	400: 	// Send mover to the next station
			fMoverPosition     := fNextStationWaitingPosition;
			fMoverVelocity     :=    300.0;
			fMoverAcceleration :=  1_000.0;
			fMoverJerk         := 10_000.0;	
	
			stMoveParameters.direction := Tc3_Mc3PlanarMotion.MC_DIRECTION.mcDirectionPositive;
			stMoveParameters.gap       := 240.0;
			
			strInfo := CONCAT('Station: ', UINT_TO_STRING(nStationIndex));
			strInfo := CONCAT(strInfo, ' Mover: ');
			strInfo := CONCAT(strInfo, UDINT_TO_STRING(nMoverIndex));
			strInfo := CONCAT(strInfo, ' move to next Station:' );
			strInfo := CONCAT(strInfo, UDINT_TO_STRING(nNextStationIndex));
			
		
			IF NOT ipMoverApplication[nMoverIndex].std.P_MoveOnTrack.Busy THEN
	
				FOR idx:=10 TO 1 BY -1 DO 
					strInfoHistory[idx] := strInfoHistory[idx-1];
				END_FOR
				strInfoHistory[0] := strInfo;		
			
				ipMoverApplication[nMoverIndex].std.MoveOnTrack( strInfo,
																 ipTrack[nNextStationTrackIndex].std,
																 fMoverPosition,
																 fMoverVelocity,
																 fMoverAcceleration,
																 fMoverJerk,
																 stMoveParameters.gap,
																 stMoveParameters.direction);
				nStateMoverRecovery := nStateMoverRecovery +1;
				
				
				ipMoverApplication[nMoverIndex].ProductData.bInitRun            := TRUE;
				ipMoverApplication[nMoverIndex].ProductData.nDestinationProcess := 0;
			END_IF	
			
	401: 
		IF ipMoverApplication[nMoverIndex].std.P_MoveOnTrack.Active THEN
			nStateMoverRecovery := 410;
		 END_IF
				 
	410: // Mover to the list of the next station
		ipStation[nNextStationIndex].P_List.AddMover(fbInitList.RemoveFirstInList());
		nStateMoverRecovery := 300;	
	
	500:	// Mover recovery done
			  MoverRecovery := TRUE;
		nStateMoverRecovery := 0;		

END_CASE
END_METHOD

PROPERTY P_bMoverError : BOOL
GET
P_bMoverError := bMoverError;
END_GET
SET
bMoverError := P_bMoverError;
END_SET
END_PROPERTY

PROPERTY PUBLIC P_nAbortingSequence : UDINT
GET
P_nAbortingSequence := nAbortingSequence;
END_GET
END_PROPERTY

PROPERTY PUBLIC P_nExecutingSequence : UDINT
GET
P_nExecutingSequence := nExecutingSequence;
END_GET
END_PROPERTY

PROPERTY PUBLIC P_nResettingSequence : UDINT
GET
P_nResettingSequence := nResettingSequence;
END_GET
END_PROPERTY

PROPERTY PUBLIC P_nStartingSequence : UDINT
GET
P_nStartingSequence := nStartingSequence;
END_GET
END_PROPERTY

PROPERTY PUBLIC P_nStartupSequence : UDINT
GET
P_nStartupSequence := nStartupSequence;
END_GET
END_PROPERTY

METHOD Resetting : BOOL
VAR_INPUT
END_VAR
CASE nResettingSequence OF 
	
	0: //Idle 
		nResettingSequence := 20;
		
		
	20: // Reset Movers
		IF ipMotionSystem.ResetMovers() THEN
			nResettingSequence := 21;
		ELSE
			;// Error			
		END_IF
		
	21: IF ipMotionSystem.P_ResetMovers.Done THEN
			nResettingSequence := 30;
		ELSIF ipMotionSystem.P_ResetMovers.Error THEN
			;//Error 	
		END_IF

		
	30:	nResettingSequence := 40;
		

	40: // Adding Environment to Group
		IF ipMotionSystem.AddEnvironmentToGroup() THEN
			nResettingSequence := 41;
		END_IF	
		
	41: IF ipMotionSystem.P_AddEnviromentToGroup.Done THEN
			nResettingSequence := 50;
		END_IF	
		
	
	50: // Enable all tracks
		IF ipMotionSystem.EnableTracks() THEN
			nResettingSequence := 51;
		ELSE
			nResettingSequence := 55;
		END_IF
		
	51:	
		IF ipMotionSystem.P_EnableTracks.Done THEN
			nResettingSequence := 60;
		ELSIF ipMotionSystem.P_EnableTracks.Error THEN
			;
		END_IF
			
	60: 
		IF ipMotionSystem.AddTracksToGroup() THEN
			nResettingSequence := 61;
		ELSE
			nResettingSequence := 65;
		END_IF
	
	61:
		IF ipMotionSystem.P_AddTracksToGroup.Done THEN
			nResettingSequence := 70;
		ELSIF ipMotionSystem.P_AddTracksToGroup.Error THEN
			;	
		END_IF
		
		
	70:	// Reset all Stations
		bDone := TRUE;
		FOR nForCounter := 1 TO nStationCount DO
			bDone := bDone AND ipStation[nForCounter].ResetStation(TRUE);
		END_FOR
		
		IF bDone THEN
			FOR nForCounter := 1 TO nStationCount DO
				ipStation[nForCounter].ResetStation(FALSE);
			END_FOR
			nResettingSequence := 80;
		END_IF
		
		
	80:	nResettingSequence := 100;	
		

		
	100: // Reset done
		nResettingSequence := 0; 
		         Resetting := TRUE;


END_CASE
END_METHOD

METHOD Starting : BOOL
VAR
	bAllMoversDone					: BOOL; 	
END_VAR
CASE nStartingSequence OF 
	

0:		// Idle
		nStartingSequence := 10;
		

10: 	// Enable all movers
		IF ipMotionSystem.EnableMovers() THEN
			nStartingSequence := nStartingSequence + 1;
		END_IF

11: 	IF ipMotionSystem.P_EnableMovers.Done THEN
			nStartingSequence := 20;
		ELSIF ipMotionSystem.P_EnableMovers.Error THEN
			;// Error = Not able to enable movers e.g. mover was not able to reach it's flight hight due to high payload 
		END_IF	


20: 	// Adding movers to the group
		IF ipMotionSystem.AddMoversToGroup() THEN
			nStartingSequence := nStartingSequence + 1;
		END_IF

21: 	IF ipMotionSystem.P_AddMoversToGroup.Done THEN
			nStartingSequence := 30;
		ELSIF ipMotionSystem.P_AddMoversToGroup.Error THEN
			;// Error
		END_IF	

		
30: 	// EnableGroup
		IF ipMotionSystem.EnableGroup() THEN
			nStartingSequence := nStartingSequence + 1;
		END_IF
	
31: 	IF ipMotionSystem.P_EnableGroup.Done THEN
			nStartingSequence := 40;
		ELSIF ipMotionSystem.P_EnableGroup.Error THEN
			;// Error
		END_IF	
		
		
40:		// Check if all are movers activated and in free movement 
		bAllMoversDone := TRUE;
		FOR nForCounter := 1 TO moverCount DO		
			IF ipMoverApplication[nForCounter].std.P_State       <> MC_PLANAR_STATE.Enabled
			OR ipMoverApplication[nForCounter].std.P_CommandMode <> MC_PLANAR_MOVER_COMMAND_MODE.FreeMovement 
			THEN
				bAllMoversDone := FALSE;
				EXIT;		
			END_IF
		END_FOR
		
		IF bAllMoversDone THEN
			nStartingSequence := 100;
		END_IF	

		
100:  // Mover Recovery/Sorting
		MoverRecovery(bReset:=TRUE);
		nStartingSequence := 101;	

101:	IF MoverRecovery(bReset:=FALSE) THEN
			nStartingSequence := 300;	
		END_IF

300:  // Starting sequence done
				 Starting := TRUE;			 
		nStartingSequence := 0; 
		
		
		
END_CASE
END_METHOD

METHOD Startup : BOOL
VAR
	aMoverDetectionSetup	: ARRAY[1..3] OF ST_TcIoMoverDetectionSetup;
END_VAR

VAR_INST
	
	// Tracks
	nTrackToInit			: UDINT;
	nTrackToGroup			: UDINT;

END_VAR
CASE nStartupSequence OF 
	
	0: //Idle 	
		nStartupSequence := 10;
		
	
	//  ======= TRACKS =======
			
	10: // Initialization of all tracks
		IF nTrackToInit < trackCount THEN
			nTrackToInit := nTrackToInit + 1;
			nStartupSequence := nStartupSequence +1;
		ELSE
			    nTrackToInit := 0;
			nStartupSequence := 100;
		END_IF
		
	11: IF ipTrack[nTrackToInit].Initialize(TRUE) THEN
			ipTrack[nTrackToInit].Initialize(FALSE);		
			nStartupSequence := nStartupSequence -1;
		END_IF

	100: // Start-Up Done!				
		Startup := TRUE;
		
	
END_CASE
END_METHOD

PROPERTY std : I_MotionSystem
GET
IF ipMotionSystem <> 0 THEN
	std := ipMotionSystem;	
END_IF
END_GET
SET
ipMotionSystem := std;
END_SET
END_PROPERTY

END_FUNCTION_BLOCK

// ---- 2_Application/Mover/FB_ApplicationMover.TcPOU
FUNCTION_BLOCK FB_ApplicationMover IMPLEMENTS I_MoverApplication
VAR
	ipMoverStandard	: I_XPlanarMoverStandard;
	
	stProductData	: ST_ProductData;
	
	nMoverIndex		: INT;
	
	nTrackId		: UDINT;
	
	// customer Data
	bIsLoaded		: BOOL;	
		
		
		
		
		
END_VAR

VAR_OUTPUT
	VisuPos	: MoverVector;
END_VAR

METHOD Cycle
IF std <> 0 THEN
	std.cycle();
	VisuPos := std.P_ActPosition;
END_IF
END_METHOD

PROPERTY P_nMoverIndex : INT
GET
P_nMoverIndex := nMoverIndex;
END_GET
SET
nMoverIndex := P_nMoverIndex;
END_SET
END_PROPERTY

PROPERTY P_nTrackId : UDINT
GET
P_nTrackId := nTrackId;
END_GET
SET
nTrackId := P_nTrackId;
END_SET
END_PROPERTY

PROPERTY ProductData : Reference to ST_ProductData
GET
ProductData REF= stProductData;
END_GET
SET
stProductData := ProductData;
END_SET
END_PROPERTY

PROPERTY std : I_XPlanarMoverStandard
GET
IF ipMoverStandard <> 0 THEN
	std := ipMoverStandard;	
END_IF
END_GET
SET
ipMoverStandard := std;
END_SET
END_PROPERTY

END_FUNCTION_BLOCK

// ---- 2_Application/Tracks/FB_TrackSegment_1.TcPOU
FUNCTION_BLOCK FB_TrackSegment_1 EXTENDS FB_TrackBase IMPLEMENTS I_TRACK
VAR_INPUT
END_VAR
VAR_OUTPUT
END_VAR


VAR
	



END_VAR

METHOD Initialize : BOOL
VAR_INPUT
	bExecute 			: BOOL;
	
END_VAR
VAR_INST
	nState			: INT;
	fbR_TrigExecute : R_TRIG;
	
	
	TrackTable		: ARRAY[1..maxNumTrackPoints,1..3] OF LREAL;
	nPointIndex		: INT;
	nPointIndexA	: INT;	
	nPointIndexB	: INT;	
	fTestValue		: LREAL;
	idx1, idx2		: INT;
	nStartFromTrack	: INT;
	nEndAtTrack		: INT;
	bCloseLoop		: BOOL;
		
END_VAR
fbR_TrigExecute(CLK := bExecute);
IF fbR_TrigExecute.Q AND NOT bBusy THEN
	// Check if GroupRef is there, else throw an error
		nState := 10;
		bBusy := TRUE;
		bError := FALSE;
END_IF


CASE nState OF 

	10:	// Init Track-Table
	
		// *******************************************************************
		// *** This code must be eddited according to machine/track layout ***
		// *******************************************************************
	
		nStartFromTrack	:= 0;		// 0 for the first track all others according to their predecessor!
	    	nEndAtTrack := 0;		// 0 for the first track all others according to their successor! 		
		     bCloseLoop := FALSE;	// TRUE for circular track	
			
			
		TrackTable[1,1] := 480.0;	// x-koordinate
		TrackTable[1,2] := 120.0;	// y-koordinate
		TrackTable[1,3] :=   0.0;	// c
		
		TrackTable[2,1] := 240.0;	// x-koordinate
		TrackTable[2,2] := 120.0;	// y-koordinate
		TrackTable[2,3] :=   0.0;	// c		
		
		TrackTable[3,1] := 120.0;	// x-koordinate
		TrackTable[3,2] := 240.0;	// y-koordinate
		TrackTable[3,3] :=   0.0;	// c		
	
		TrackTable[4,1] := 120.0;	// x-koordinate
		TrackTable[4,2] := 480.0;	// y-koordinate
		TrackTable[4,3] :=   0.0;	// c		
	
		TrackTable[5,1] := 240.0;	// x-koordinate
		TrackTable[5,2] := 600.0;	// y-koordinate
		TrackTable[5,3] :=   0.0;	// c		
	
		TrackTable[6,1] := 480.0;	// x-koordinate
		TrackTable[6,2] := 600.0;	// y-koordinate
		TrackTable[6,3] :=   0.0;	// c				
		
		nState := 20;
		
		
	20:	// Building the track 
		IF fbTrackStandard.BuildTrack(TrackTable, 0, 0, bCloseLoop) THEN
			nState := 30;
		END_IF
		
	30: 	
		IF fbTrackStandard.P_BuildTrack.Done THEN
			nState := 100;
		END_IF
		
					 
	100: 	// MC_Reset Done
			fTrackLength := fbTrackStandard.GetLength();
				   bBusy := FALSE;
			  Initialize := TRUE;
			
			IF NOT bExecute THEN
				Initialize := FALSE;
				    nState := 0;
			END_IF
	
END_CASE
END_METHOD

END_FUNCTION_BLOCK

// ---- 2_Application/Tracks/FB_TrackBase.TcPOU
FUNCTION_BLOCK FB_TrackBase
VAR_INPUT
END_VAR
VAR_OUTPUT
	bBusy 	: BOOL;
	bError 	: BOOL;
END_VAR
VAR
	trackLinePosStart 	: PositionXYC;
	trackLinePosEnd 	: PositionXYC;
	fbTrackStandard		: FB_TrackStandard;
	fTrackLength		: LREAL;
END_VAR

METHOD ccl00_cycle : BOOL
VAR_INPUT
END_VAR
fbTrackStandard.Cycle();
END_METHOD

PROPERTY P_TrackLength : LREAL
GET
P_TrackLength := fTrackLength;
END_GET
END_PROPERTY

PROPERTY std : I_TrackStandard
GET
std := fbTrackStandard;
END_GET
END_PROPERTY

END_FUNCTION_BLOCK

// ---- 2_Application/Tracks/FB_TrackSegment_2.TcPOU
FUNCTION_BLOCK FB_TrackSegment_2 EXTENDS FB_TrackBase IMPLEMENTS I_TRACK
VAR_INPUT
END_VAR
VAR_OUTPUT
END_VAR


VAR
	



END_VAR

METHOD Initialize : BOOL
VAR_INPUT
	bExecute 			: BOOL;
	
END_VAR
VAR_INST
	nState			: INT;
	fbR_TrigExecute : R_TRIG;
	
	
	TrackTable		: ARRAY[1..maxNumTrackPoints,1..3] OF LREAL;
	nPointIndex		: INT;
	nPointIndexA	: INT;	
	nPointIndexB	: INT;	
	fTestValue		: LREAL;
	idx1, idx2		: INT;
	nStartFromTrack	: INT;
	nEndAtTrack		: INT;
	bCloseLoop		: BOOL;
	
END_VAR
fbR_TrigExecute(CLK := bExecute);
IF fbR_TrigExecute.Q AND NOT bBusy THEN
	// Check if GroupRef is there, else throw an error
		nState := 10;
		bBusy := TRUE;
		bError := FALSE;
END_IF



CASE nState OF 

	10:	// Init Track-Table
	
		// *******************************************************************
		// *** This code must be eddited according to machine/track layout ***
		// *******************************************************************
	
		nStartFromTrack	:= 1;		// 0 for the first track all others according to their predecessor!
	    	nEndAtTrack := 1;		// 0 for the first track all others according to their successor! 		
			 bCloseLoop := FALSE;	// TRUE for circular track	
		
		TrackTable[1,1] := 600.0;	// x-koordinate
		TrackTable[1,2] := 480.0;	// y-koordinate
		TrackTable[1,3] :=   0.0;	// c
		
		TrackTable[2,1] := 600.0;	// x-koordinate
		TrackTable[2,2] := 240.0;	// y-koordinate
		TrackTable[2,3] :=   0.0;	// c		

		TrackTable[3,1] :=   0.0;	// x-koordinate
		TrackTable[3,2] :=   0.0;	// y-koordinate
		TrackTable[3,3] :=   0.0;	// c		
	
		TrackTable[4,1] :=   0.0;	// x-koordinate
		TrackTable[4,2] :=   0.0;	// y-koordinate
		TrackTable[4,3] :=   0.0;	// c		
	
		TrackTable[5,1] :=   0.0;	// x-koordinate
		TrackTable[5,2] :=   0.0;	// y-koordinate
		TrackTable[5,3] :=   0.0;	// c		
	
		TrackTable[6,1] :=   0.0;	// x-koordinate
		TrackTable[6,2] :=   0.0;	// y-koordinate
		TrackTable[6,3] :=   0.0;	// c				

		TrackTable[7,1] :=   0.0;	// x-koordinate
		TrackTable[7,2] :=   0.0;	// y-koordinate
		TrackTable[7,3] :=   0.0;	// c		
	
		TrackTable[8,1] :=   0.0;	// x-koordinate
		TrackTable[8,2] :=   0.0;	// y-koordinate
		TrackTable[8,3] :=   0.0;	// c	

		
		nState := 20;
		
	20:	// Building the track 
		IF fbTrackStandard.BuildTrack(TrackTable, ipTrack[1].std, ipTrack[1].std, bCloseLoop) THEN
			nState := 30;
		END_IF		
	30: 	
		IF fbTrackStandard.P_BuildTrack.Done THEN
			nState := 100;
		END_IF
		
					 
	100: 	// MC_Reset Done
			fTrackLength := fbTrackStandard.GetLength();
				   bBusy := FALSE;
			  Initialize := TRUE;
			
			IF NOT bExecute THEN
				Initialize := FALSE;
				    nState := 0;
			END_IF
	
END_CASE
END_METHOD

END_FUNCTION_BLOCK

// ---- 2_Application/Tracks/FB_TrackSegment_3.TcPOU
FUNCTION_BLOCK FB_TrackSegment_3 EXTENDS FB_TrackBase IMPLEMENTS I_TRACK
VAR_INPUT
END_VAR
VAR_OUTPUT
END_VAR


VAR
	



END_VAR

METHOD Initialize : BOOL
VAR_INPUT
	bExecute 			: BOOL;
	
END_VAR
VAR_INST
	nState			: INT;
	fbR_TrigExecute : R_TRIG;
	
	
	TrackTable		: ARRAY[1..maxNumTrackPoints,1..3] OF LREAL;
	nPointIndex		: INT;
	nPointIndexA	: INT;	
	nPointIndexB	: INT;	
	fTestValue		: LREAL;
	idx1, idx2		: INT;
	nStartFromTrack	: INT;
	nEndAtTrack		: INT;
	bCloseLoop		: BOOL;
	
END_VAR
fbR_TrigExecute(CLK := bExecute);
IF fbR_TrigExecute.Q AND NOT bBusy THEN
	// Check if GroupRef is there, else throw an error
		nState := 10;
		bBusy := TRUE;
		bError := FALSE;
END_IF



CASE nState OF 

	10:	// Init Track-Table
	
		// *******************************************************************
		// *** This code must be eddited according to machine/track layout ***
		// *******************************************************************
	
		nStartFromTrack	:= 1;		// 0 for the first track all others according to their predecessor!
	    	nEndAtTrack := 1;		// 0 for the first track all others according to their successor! 		
			 bCloseLoop := FALSE;	// TRUE for circular track		
	
		TrackTable[1,1] := 480.0;	// x-koordinate
		TrackTable[1,2] := 600.0;	// y-koordinate
		TrackTable[1,3] :=   0.0;	// c
		
		TrackTable[2,1] := 720.0;	// x-koordinate
		TrackTable[2,2] := 600.0;	// y-koordinate
		TrackTable[2,3] :=   0.0;	// c		
		
		TrackTable[3,1] := 840.0;	// x-koordinate
		TrackTable[3,2] := 480.0;	// y-koordinate
		TrackTable[3,3] :=   0.0;	// c		
	
		TrackTable[4,1] := 840.0;	// x-koordinate
		TrackTable[4,2] := 240.0;	// y-koordinate
		TrackTable[4,3] :=   0.0;	// c		
	
		TrackTable[5,1] := 720.0;	// x-koordinate
		TrackTable[5,2] := 120.0;	// y-koordinate
		TrackTable[5,3] :=   0.0;	// c		
	
		TrackTable[6,1] := 480.0;	// x-koordinate
		TrackTable[6,2] := 120.0;	// y-koordinate
		TrackTable[6,3] :=   0.0;	// c			
			
		nState := 20;

	20:	// Building the track 
		IF fbTrackStandard.BuildTrack(TrackTable, ipTrack[1].std, ipTrack[1].std, bCloseLoop) THEN
			nState := 30;
		END_IF
		
	30: 	
		IF fbTrackStandard.P_BuildTrack.Done THEN
			nState := 100;
		END_IF
		
					 
	100: 	// MC_Reset Done
			fTrackLength := fbTrackStandard.GetLength();
				   bBusy := FALSE;
			  Initialize := TRUE;
			
			IF NOT bExecute THEN
				Initialize := FALSE;
				    nState := 0;
			END_IF
	
END_CASE
END_METHOD

END_FUNCTION_BLOCK

// ---- 2_Application/Station/FB_Station_01_Process.TcPOU
FUNCTION_BLOCK FB_Station_01_Process EXTENDS FB_StationBase
VAR_INPUT
END_VAR
VAR_OUTPUT
END_VAR
VAR
END_VAR

METHOD ClearList : BOOL
VAR_INPUT
END_VAR
SUPER^.ClearList();
// Add aditional Data to Clear in Reset
// List and State will be cleared in master class
ClearList := TRUE;
END_METHOD

METHOD Processing : BOOL
VAR_INPUT
	i_nMachineState 	: INT;		// 1=starting, 2=Running
END_VAR



VAR_INST

	bToggleSwitch	: BOOL;
	bStationActive				: BOOL;

	nMoverIndex					: UINT;
	fPositionOnTrack			: LREAL;
	nCurrentTrackIndex			: UDINT;
	
	nStationIndex				: UINT;
	nNextStationIndex			: UINT;
	nStationTrackIndex			: UINT;
	fStationPositionOnTrack		: LREAL;
	fSendAwayPosition			: LREAL;
	fInRangePosition			: LREAL;
	fOutOfRangePosition			: LREAL;
	
	fMoverPosition				: LREAL;
	nTrackIndex					: UINT;
	fMoverVelocity				: LREAL;
	fMoverAcceleration			: LREAL;
	fMoverJerk					: LREAL;
	strInfo						: STRING;
	
	nErrorId					: UDINT;
	nObjectID					: UDINT;
	nObjectType					: UDINT;						
	
	Timer01						: TON;
	ClearTrig					: R_TRIG;
	
	TrackInfo					: PlanarObjectInfo;
	nStationTrackID				: UDINT;
	nMoverOnTrackID				: UDINT;
	
END_VAR


// *** Processing Station ***

ClearTrig(CLK:=bClearStation);
IF ClearTrig.Q THEN
	nState := 10;	
END_IF


CASE nState OF

	0:		// Waiting for initialization	
			nState := 10;

	10:		// Init Station-Parameters				
				      nStationIndex := 1;	
			     nStationTrackIndex := 1;
			      nNextStationIndex := 4;
			fStationPositionOnTrack := ipTrack[nStationTrackIndex].P_TrackLength/2.0;
				  fSendAwayPosition := ipTrack[nStationTrackIndex].P_TrackLength - 120.0; 		
										
			bClearStation := FALSE;
				   nState := 11;

	11: // Fail-safe check, just to make sure all variables have been assigned after doing copy&paste from the template
			IF            nStationIndex > 0
			AND      nStationTrackIndex > 0
			AND       nNextStationIndex > 0
			AND fStationPositionOnTrack > 0
			AND       fSendAwayPosition > 0
			THEN   
				nState := 20;
			END_IF
			
				   
	20:		// Calculating station x-y-position 
			PositionOnTrack.fPositionOnTrack := fStationPositionOnTrack;
 			PositionOnTrack.nTrackId		 := UINT_TO_INT(nStationTrackIndex);
			ipTrack[PositionOnTrack.nTrackId].std.GetMoverPositionAt(PositionOnTrack.fPositionOnTrack, StationPosition);
			VisuPosX := StationPosition.x;
			VisuPosY := StationPosition.y;
			nState := 100;

		
	100: 	// Waiting for Mover
			IF P_List.P_FirstInList <> 0 THEN
					   nMoverIndex := P_List.P_FirstInList.P_Id;
							nState := 110;
			END_IF
	
		
	110: 	// Check if Mover is in range
			TrackInfo := ipTrack[nStationTrackIndex].std.P_Info;
			nStationTrackID := TrackInfo.Id;
			nMoverOnTrackID := ipMoverApplication[nMoverIndex].std.P_SetOnTrack.TrackOID;
			IF nStationTrackID = nMoverOnTrackID  THEN
				nCurrentTrackIndex := nMoverOnTrackID;
							nState := 120;		
			ELSE
				nState := 100;
			END_IF
		
		
	120: 	// Checking product properties
			IF i_nMachineState = 1  THEN    // 1=starting, 2=Running
				IF nStationIndex = 1 THEN
					ipMoverApplication[nMoverIndex].ProductData.bInitRun := FALSE;
				ELSE
					nState := 220;
				END_IF
			ELSIF i_nMachineState = 2 THEN  // 1=starting, 2=Running
				nState := 200;
			ELSE
				nState := 20;	
			END_IF			
		
		
	200: 	// Send mover to Processing-Position
			fMoverPosition     := fStationPositionOnTrack;
			nTrackIndex        := nStationTrackIndex;
			fMoverVelocity     :=    300.0;
			fMoverAcceleration :=  1_000.0;
			fMoverJerk         := 10_000.0;	
	
			stMoveParameters.direction := Tc3_Mc3PlanarMotion.MC_DIRECTION.mcDirectionPositive;
			stMoveParameters.gap       := 240.0;
		
			strInfo := CONCAT('Station: ', UINT_TO_STRING(nStationIndex));
			strInfo := CONCAT(strInfo, ' to processing position');

			
			IF NOT ipMoverApplication[nMoverIndex].std.P_MoveOnTrack.Error THEN
	
				FOR idx:=10 TO 1 BY -1 DO 
					strInfoHistory[idx] := strInfoHistory[idx-1];
				END_FOR
				strInfoHistory[0] := strInfo;		

	
				ipMoverApplication[nMoverIndex].std.MoveOnTrack( strInfo,
																 ipTrack[nTrackIndex].std,
																 fMoverPosition,
																 fMoverVelocity,
																 fMoverAcceleration,
																 fMoverJerk,
																 stMoveParameters.gap,
																 stMoveParameters.direction);
				nState := nState +1;
				
			ELSIF ipMoverApplication[nMoverIndex].std.P_MoveOnTrack.Error THEN
				   nErrorID := ipMoverApplication[nMoverIndex].std.P_MoveOnTrack.ErrorID;
				  nObjectID := ipMoverApplication[nMoverIndex].std.P_MoveOnTrack.stInfo.nObjectID;
				nObjectType := ipMoverApplication[nMoverIndex].std.P_MoveOnTrack.stInfo.nObjectType;				
			END_IF
		
		
	201: 	IF ipMoverApplication[nMoverIndex].std.P_MoveOnTrack.Done THEN
				nState := 210;
			ELSIF ipMoverApplication[nMoverIndex].std.P_MoveOnTrack.Error THEN
				   nErrorID := ipMoverApplication[nMoverIndex].std.P_MoveOnTrack.ErrorID;
				  nObjectID := ipMoverApplication[nMoverIndex].std.P_MoveOnTrack.stInfo.nObjectID;
				nObjectType := ipMoverApplication[nMoverIndex].std.P_MoveOnTrack.stInfo.nObjectType;
			END_IF		
		
		
	210: 	// do process
			Timer01(IN:=TRUE, PT:=T#1S);
			IF Timer01.Q THEN
				Timer01(IN:=FALSE);	
						
				IF nStationIndex = 1 THEN	
					// Station 1 toggeling mover destination to Station2 or Station3
					IF bToggleSwitch THEN
						ipMoverApplication[nMoverIndex].ProductData.nDestinationProcess := 2;
					ELSE
						ipMoverApplication[nMoverIndex].ProductData.nDestinationProcess := 3;		
					END_IF
					bToggleSwitch := NOT bToggleSwitch;					
				ELSE
					ipMoverApplication[nMoverIndex].ProductData.nDestinationProcess := 1;
				END_IF	
				
				nState := 220;
			END_IF

		
	220: 	// Send mover to the next station
			fMoverPosition     := fSendAwayPosition;	
			nTrackIndex        := nStationTrackIndex;		
			fMoverVelocity     :=    300.0;
			fMoverAcceleration :=  1_000.0;
			fMoverJerk         := 10_000.0;	
	
			stMoveParameters.direction := Tc3_Mc3PlanarMotion.MC_DIRECTION.mcDirectionPositive;
			stMoveParameters.gap       := 240.0;
			
			strInfo := CONCAT('Station: ', UINT_TO_STRING(nStationIndex));
			strInfo := CONCAT(strInfo, ' move to next Station:' );
			strInfo := CONCAT(strInfo, UINT_TO_STRING(nNextStationIndex));

			
			IF ipMoverApplication[nMoverIndex].std.P_MoveOnTrack.Done THEN

				FOR idx:=10 TO 1 BY -1 DO 
					strInfoHistory[idx] := strInfoHistory[idx-1];
				END_FOR
				strInfoHistory[0] := strInfo;		
			
				ipMoverApplication[nMoverIndex].std.MoveOnTrack( strInfo,
																 ipTrack[nTrackIndex].std,
																 fMoverPosition,
																 fMoverVelocity,
																 fMoverAcceleration,
																 fMoverJerk,
																 stMoveParameters.gap,
																 stMoveParameters.direction);
				nState := nState +1;
			END_IF		
		
		
	221: 	IF ipMoverApplication[nMoverIndex].std.P_MoveOnTrack.Active
			OR ipMoverApplication[nMoverIndex].std.P_MoveOnTrack.Done 
			THEN
				nState := 230;
			ELSIF ipMoverApplication[nMoverIndex].std.P_MoveOnTrack.Error THEN
				
				   nErrorID := ipMoverApplication[nMoverIndex].std.P_MoveOnTrack.ErrorID;
				  nObjectID := ipMoverApplication[nMoverIndex].std.P_MoveOnTrack.stInfo.nObjectID;
				nObjectType := ipMoverApplication[nMoverIndex].std.P_MoveOnTrack.stInfo.nObjectType;
			END_IF		
		
			
	230: 	// Mover to the list of the next station
			ipStation[nNextStationIndex].P_List.AddMover(P_List.RemoveFirstInList());
			nState := 500;	
	
		
	500: 	// Done for this cycle
			nState := 100;

END_CASE
END_METHOD

END_FUNCTION_BLOCK

// ---- 2_Application/Station/FB_StationBase.TcPOU
FUNCTION_BLOCK FB_StationBase IMPLEMENTS I_Station
VAR
	stMoveParameters 	: ST_MoveOnTrackOptions; 		
END_VAR
VAR_OUTPUT
	VisuPosX			: LREAL;
	VisuPosY			: LREAL;
END_VAR

VAR

	idx  				: UDINT;
	nState 				: INT;	
	nStateInit			: INT;
	
	StationPosition     : PositionXYC;	
	PositionOnTrack		: ST_StationTrackPosition;

	ipMoverInStation	: I_MoverApplication;
	ipListAhead 		: I_List;

	fbList_Station		: FB_List;
	fbList_InputB		: FB_List;	
	fbList_InputC		: FB_List;		
	
	bClearStation		: BOOL;

	strInfo				: STRING;
	strInfoHistory		: ARRAY[0..10] OF STRING;
	
	nErrorCode			: UDINT;

END_VAR

METHOD ccl00_cycle : BOOL
VAR_INPUT
END_VAR
VAR
	nForCounter : INT;
END_VAR


VAR_INST
	
	fTestValueX	: LREAL;
	fTestValueY : LREAL;	
	
END_VAR



;
END_METHOD

METHOD ClearList : BOOL
VAR_INPUT
END_VAR



	fbList_Station.ClearList();
	ClearList := TRUE;
END_METHOD

PROPERTY InputConnections : I_Station
GET
END_GET
SET
END_SET
END_PROPERTY

PROPERTY OutputConnections : I_Station
GET
END_GET
SET
END_SET
END_PROPERTY

PROPERTY P_List : I_List
GET
P_List := fbList_Station;
END_GET
END_PROPERTY

PROPERTY P_List_Input_B : I_List
GET
P_List_Input_B := fbList_InputB;
END_GET
END_PROPERTY

PROPERTY P_List_Input_C : I_List
GET
P_List_Input_C := fbList_InputC;
END_GET
END_PROPERTY

PROPERTY P_nErrorCode : UDINT
GET
P_nErrorCode := nErrorCode;
END_GET
END_PROPERTY

PROPERTY P_Position : BOOL //PositionXYC
GET
//P_Position := StationPosition;
END_GET
END_PROPERTY

PROPERTY P_PositionOnTrack : ST_StationTrackPosition
GET
P_PositionOnTrack := PositionOnTrack;
END_GET
END_PROPERTY

METHOD Processing : BOOL
VAR_INPUT
	i_nMachineState 	: INT;		// 1=Starting, 2=Running
END_VAR

CASE nState OF
	
	0: // waiting for Mover
	
	
	10: // do process
	
	100: // mover mover to nother list


END_CASE
END_METHOD

METHOD ResetStation : BOOL
VAR_INPUT
	bClear	: BOOL;
END_VAR


VAR_INST
	nStateReset : INT;	
	nTestCnt	: INT;
END_VAR


	CASE nStateReset OF
		
	0:	IF bClear THEN
			ResetStation := FALSE;
			 nStateReset := 10;
		END_IF
	
	10: 
		bClearStation := TRUE;
		nState := 0;
		IF ClearList() THEN 
			nStateReset := 20;
		END_IF
		nTestCnt := nTestCnt +1;
	
	20:	
		ResetStation := TRUE;
		 nStateReset := 30;
		 
	30: 
		IF NOT bClear THEN
			nStateReset := 0;
		END_IF 
		
	END_CASE
END_METHOD

END_FUNCTION_BLOCK

// ---- 2_Application/Station/FB_Station_02_Process.TcPOU
FUNCTION_BLOCK FB_Station_02_Process EXTENDS FB_StationBase
VAR_INPUT
END_VAR
VAR_OUTPUT
END_VAR
VAR
END_VAR

METHOD ClearList : BOOL
VAR_INPUT
END_VAR
SUPER^.ClearList();
// Add aditional Data to Clear in Reset
// List and State will be cleared in master class
ClearList := TRUE;
END_METHOD

METHOD Processing : BOOL
VAR_INPUT
	i_nMachineState 	: INT;		// 1=starting, 2=Running
END_VAR



VAR_INST

	bToggleSwitch	: BOOL;
	bStationActive				: BOOL;

	nMoverIndex					: UINT;
	fPositionOnTrack			: LREAL;
	nCurrentTrackIndex			: UDINT;
	
	nStationIndex				: UINT;
	nNextStationIndex			: UINT;
	nStationTrackIndex			: UINT;
	fStationPositionOnTrack		: LREAL;
	fSendAwayPosition			: LREAL;
	fInRangePosition			: LREAL;
	fOutOfRangePosition			: LREAL;
	
	fMoverPosition				: LREAL;
	nTrackIndex					: UINT;
	fMoverVelocity				: LREAL;
	fMoverAcceleration			: LREAL;
	fMoverJerk					: LREAL;
	strInfo						: STRING;
	
	nErrorId					: UDINT;
	nObjectID					: UDINT;
	nObjectType					: UDINT;						
	
	Timer01						: TON;
	ClearTrig					: R_TRIG;
	
	TrackInfo				: PlanarObjectInfo;
	nStationTrackID			: UDINT;
	nMoverOnTrackID			: UDINT;
	
END_VAR


// *** Processing Station ***




ClearTrig(CLK:=bClearStation);
IF ClearTrig.Q THEN
	nState := 10;	
END_IF




CASE nState OF


	0:		// Waiting for initialization	
			nState := 10;
	
		
	10:		// Init Station-Parameters					
				      nStationIndex := 2;	
			     nStationTrackIndex := 2;
			      nNextStationIndex := 5;
			fStationPositionOnTrack := ipTrack[nStationTrackIndex].P_TrackLength/2.0;
		          fSendAwayPosition := fStationPositionOnTrack + 10.0; 	
												
			bClearStation := FALSE;
				   nState := 11;

	11: // Fail-safe check, just to make sure all variables have been assigned after doing copy&paste from the template
			IF            nStationIndex > 0
			AND      nStationTrackIndex > 0
			AND       nNextStationIndex > 0
			AND fStationPositionOnTrack > 0
			AND       fSendAwayPosition > 0
			THEN   
				nState := 20;
			END_IF
	
				   
	20:		// Calculating station x-y-position 
			PositionOnTrack.fPositionOnTrack := fStationPositionOnTrack;
 			PositionOnTrack.nTrackId		 := UINT_TO_INT(nStationTrackIndex);
			ipTrack[PositionOnTrack.nTrackId].std.GetMoverPositionAt(PositionOnTrack.fPositionOnTrack, StationPosition);
			VisuPosX := StationPosition.x;
			VisuPosY := StationPosition.y;
			nState := 100;

		
		100: 	// Waiting for Mover
			IF P_List.P_FirstInList <> 0 THEN
					   nMoverIndex := P_List.P_FirstInList.P_Id;
							nState := 110;
			END_IF
	
		
	110: 	// Check if Mover is in range
			TrackInfo := ipTrack[nStationTrackIndex].std.P_Info;
			nStationTrackID := TrackInfo.Id;
			nMoverOnTrackID := ipMoverApplication[nMoverIndex].std.P_SetOnTrack.TrackOID;
			IF nStationTrackID = nMoverOnTrackID  THEN
				nCurrentTrackIndex := nMoverOnTrackID;
							nState := 120;		
			ELSE
				nState := 100;
			END_IF
		
		
	120: 	// Checking product properties
			IF i_nMachineState = 1  THEN    // 1=starting, 2=Running
				IF nStationIndex = 1 THEN
					ipMoverApplication[nMoverIndex].ProductData.bInitRun := FALSE;
				ELSE
					nState := 220;
				END_IF
			ELSIF i_nMachineState = 2 THEN  // 1=starting, 2=Running
				nState := 200;
			ELSE
				nState := 20;	
			END_IF			
		
		
	200: 	// Send mover to Processing-Position
			fMoverPosition     := fStationPositionOnTrack;
			nTrackIndex        := nStationTrackIndex;
			fMoverVelocity     :=    300.0;
			fMoverAcceleration :=  1_000.0;
			fMoverJerk         := 10_000.0;	
	
			stMoveParameters.direction := Tc3_Mc3PlanarMotion.MC_DIRECTION.mcDirectionPositive;
			stMoveParameters.gap       := 240.0;
		
			strInfo := CONCAT('Station: ', UINT_TO_STRING(nStationIndex));
			strInfo := CONCAT(strInfo, ' to processing position');

			
			IF NOT ipMoverApplication[nMoverIndex].std.P_MoveOnTrack.Error THEN
	
				FOR idx:=10 TO 1 BY -1 DO 
					strInfoHistory[idx] := strInfoHistory[idx-1];
				END_FOR
				strInfoHistory[0] := strInfo;		

	
				ipMoverApplication[nMoverIndex].std.MoveOnTrack( strInfo,
																 ipTrack[nTrackIndex].std,
																 fMoverPosition,
																 fMoverVelocity,
																 fMoverAcceleration,
																 fMoverJerk,
																 stMoveParameters.gap,
																 stMoveParameters.direction);
				nState := nState +1;
				
			ELSIF ipMoverApplication[nMoverIndex].std.P_MoveOnTrack.Error THEN
				   nErrorID := ipMoverApplication[nMoverIndex].std.P_MoveOnTrack.ErrorID;
				  nObjectID := ipMoverApplication[nMoverIndex].std.P_MoveOnTrack.stInfo.nObjectID;
				nObjectType := ipMoverApplication[nMoverIndex].std.P_MoveOnTrack.stInfo.nObjectType;				
			END_IF
		
		
	201: 	IF ipMoverApplication[nMoverIndex].std.P_MoveOnTrack.Done THEN
				nState := 210;
			ELSIF ipMoverApplication[nMoverIndex].std.P_MoveOnTrack.Error THEN
				   nErrorID := ipMoverApplication[nMoverIndex].std.P_MoveOnTrack.ErrorID;
				  nObjectID := ipMoverApplication[nMoverIndex].std.P_MoveOnTrack.stInfo.nObjectID;
				nObjectType := ipMoverApplication[nMoverIndex].std.P_MoveOnTrack.stInfo.nObjectType;
			END_IF		
		
		
	210: 	// do process
			Timer01(IN:=TRUE, PT:=T#1S);
			IF Timer01.Q THEN
				Timer01(IN:=FALSE);	
						
				IF nStationIndex = 1 THEN	
					// Station 1 toggeling mover destination to Station2 or Station3
					IF bToggleSwitch THEN
						ipMoverApplication[nMoverIndex].ProductData.nDestinationProcess := 2;
					ELSE
						ipMoverApplication[nMoverIndex].ProductData.nDestinationProcess := 3;		
					END_IF
					bToggleSwitch := NOT bToggleSwitch;					
				ELSE
					ipMoverApplication[nMoverIndex].ProductData.nDestinationProcess := 1;
				END_IF	
				
				nState := 220;
			END_IF

		
	220: 	// Send mover to the next station
			fMoverPosition     := fSendAwayPosition;	
			nTrackIndex        := nStationTrackIndex;		
			fMoverVelocity     :=    300.0;
			fMoverAcceleration :=  1_000.0;
			fMoverJerk         := 10_000.0;	
	
			stMoveParameters.direction := Tc3_Mc3PlanarMotion.MC_DIRECTION.mcDirectionPositive;
			stMoveParameters.gap       := 240.0;
			
			strInfo := CONCAT('Station: ', UINT_TO_STRING(nStationIndex));
			strInfo := CONCAT(strInfo, ' move to next Station:' );
			strInfo := CONCAT(strInfo, UINT_TO_STRING(nNextStationIndex));

			
			IF ipMoverApplication[nMoverIndex].std.P_MoveOnTrack.Done THEN

				FOR idx:=10 TO 1 BY -1 DO 
					strInfoHistory[idx] := strInfoHistory[idx-1];
				END_FOR
				strInfoHistory[0] := strInfo;		
			
				ipMoverApplication[nMoverIndex].std.MoveOnTrack( strInfo,
																 ipTrack[nTrackIndex].std,
																 fMoverPosition,
																 fMoverVelocity,
																 fMoverAcceleration,
																 fMoverJerk,
																 stMoveParameters.gap,
																 stMoveParameters.direction);
				nState := nState +1;
			END_IF		
		
		
	221: 	IF ipMoverApplication[nMoverIndex].std.P_MoveOnTrack.Active
			OR ipMoverApplication[nMoverIndex].std.P_MoveOnTrack.Done 
			THEN
				nState := 230;
			ELSIF ipMoverApplication[nMoverIndex].std.P_MoveOnTrack.Error THEN
				
				   nErrorID := ipMoverApplication[nMoverIndex].std.P_MoveOnTrack.ErrorID;
				  nObjectID := ipMoverApplication[nMoverIndex].std.P_MoveOnTrack.stInfo.nObjectID;
				nObjectType := ipMoverApplication[nMoverIndex].std.P_MoveOnTrack.stInfo.nObjectType;
			END_IF		
		
			
	230: 	// Mover to the list of the next station
			ipStation[nNextStationIndex].P_List.AddMover(P_List.RemoveFirstInList());
			nState := 500;	
	
		
	500: 	// Done for this cycle
			nState := 100;

END_CASE
END_METHOD

END_FUNCTION_BLOCK

// ---- 2_Application/Station/FB_Station_03_Process.TcPOU
FUNCTION_BLOCK FB_Station_03_Process EXTENDS FB_StationBase
VAR_INPUT
END_VAR
VAR_OUTPUT
END_VAR
VAR
END_VAR

METHOD ClearList : BOOL
VAR_INPUT
END_VAR
SUPER^.ClearList();
// Add aditional Data to Clear in Reset
// List and State will be cleared in master class
ClearList := TRUE;
END_METHOD

METHOD Processing : BOOL
VAR_INPUT
	i_nMachineState 	: INT;		// 1=starting, 2=Running
END_VAR



VAR_INST

	bToggleSwitch	: BOOL;

	nMoverIndex					: UINT;
	fPositionOnTrack			: LREAL;
	nCurrentTrackIndex			: UDINT;
	
	nStationIndex				: UINT;
	nNextStationIndex			: UINT;
	nStationTrackIndex			: UINT;
	fStationPositionOnTrack		: LREAL;
	fSendAwayPosition			: LREAL;
	fInRangePosition			: LREAL;
	fOutOfRangePosition			: LREAL;
	
	fMoverPosition				: LREAL;
	nTrackIndex					: UINT;
	fMoverVelocity				: LREAL;
	fMoverAcceleration			: LREAL;
	fMoverJerk					: LREAL;
	strInfo						: STRING;
	
	nErrorId					: UDINT;
	nObjectID					: UDINT;
	nObjectType					: UDINT;						
	
	Timer01						: TON;
	ClearTrig					: R_TRIG;
	
	TrackInfo					: PlanarObjectInfo;
	nStationTrackID				: UDINT;
	nMoverOnTrackID				: UDINT;
	
END_VAR


// *** Processing Station ***


ClearTrig(CLK:=bClearStation);
IF ClearTrig.Q THEN
	nState := 10;	
END_IF




CASE nState OF


	0:		// Waiting for initialization
			nState := 10;
		
	
	10:		// Init Station-Parameters				
				      nStationIndex := 3;	
			     nStationTrackIndex := 3;
			      nNextStationIndex := 5;  
			fStationPositionOnTrack := ipTrack[nStationTrackIndex].P_TrackLength/2.0;
			      fSendAwayPosition := fStationPositionOnTrack + 220.0; 
			
			bClearStation := FALSE;
				   nState := 11;

	11: // Fail-safe check, just to make sure all variables have been assigned after doing copy&paste from the template
			IF            nStationIndex > 0
			AND      nStationTrackIndex > 0
			AND       nNextStationIndex > 0
			AND fStationPositionOnTrack > 0
			AND       fSendAwayPosition > 0
			THEN   
				nState := 20;
			END_IF

 
	20:		// Calculating station x-y-position 
			PositionOnTrack.fPositionOnTrack := fStationPositionOnTrack;
 			PositionOnTrack.nTrackId		 := UINT_TO_INT(nStationTrackIndex);
			ipTrack[PositionOnTrack.nTrackId].std.GetMoverPositionAt(PositionOnTrack.fPositionOnTrack, StationPosition);
			VisuPosX := StationPosition.x;
			VisuPosY := StationPosition.y;
			nState := 100;

			
	100: 	// Waiting for Mover
			IF P_List.P_FirstInList <> 0 THEN
					   nMoverIndex := P_List.P_FirstInList.P_Id;
							nState := 110;
			END_IF
	
		
	110: 	// Check if Mover is in range
			TrackInfo := ipTrack[nStationTrackIndex].std.P_Info;
			nStationTrackID := TrackInfo.Id;
			nMoverOnTrackID := ipMoverApplication[nMoverIndex].std.P_SetOnTrack.TrackOID;
			IF nStationTrackID = nMoverOnTrackID  THEN
				nCurrentTrackIndex := nMoverOnTrackID;
							nState := 120;		
			ELSE
				nState := 100;
			END_IF
		
		
	120: 	// Checking product properties
			IF i_nMachineState = 1  THEN    // 1=starting, 2=Running
				IF nStationIndex = 1 THEN
					ipMoverApplication[nMoverIndex].ProductData.bInitRun := FALSE;
				ELSE
					nState := 220;
				END_IF
			ELSIF i_nMachineState = 2 THEN  // 1=starting, 2=Running
				nState := 200;
			ELSE
				nState := 20;	
			END_IF			
		
		
	200: 	// Send mover to Processing-Position
			fMoverPosition     := fStationPositionOnTrack;
			nTrackIndex        := nStationTrackIndex;
			fMoverVelocity     :=    300.0;
			fMoverAcceleration :=  1_000.0;
			fMoverJerk         := 10_000.0;	
	
			stMoveParameters.direction := Tc3_Mc3PlanarMotion.MC_DIRECTION.mcDirectionPositive;
			stMoveParameters.gap       := 240.0;
		
			strInfo := CONCAT('Station: ', UINT_TO_STRING(nStationIndex));
			strInfo := CONCAT(strInfo, ' to processing position');

			
			IF NOT ipMoverApplication[nMoverIndex].std.P_MoveOnTrack.Error THEN
	
				FOR idx:=10 TO 1 BY -1 DO 
					strInfoHistory[idx] := strInfoHistory[idx-1];
				END_FOR
				strInfoHistory[0] := strInfo;		

	
				ipMoverApplication[nMoverIndex].std.MoveOnTrack( strInfo,
																 ipTrack[nTrackIndex].std,
																 fMoverPosition,
																 fMoverVelocity,
																 fMoverAcceleration,
																 fMoverJerk,
																 stMoveParameters.gap,
																 stMoveParameters.direction);
				nState := nState +1;
				
			ELSIF ipMoverApplication[nMoverIndex].std.P_MoveOnTrack.Error THEN
				   nErrorID := ipMoverApplication[nMoverIndex].std.P_MoveOnTrack.ErrorID;
				  nObjectID := ipMoverApplication[nMoverIndex].std.P_MoveOnTrack.stInfo.nObjectID;
				nObjectType := ipMoverApplication[nMoverIndex].std.P_MoveOnTrack.stInfo.nObjectType;				
			END_IF
		
		
	201: 	IF ipMoverApplication[nMoverIndex].std.P_MoveOnTrack.Done THEN
				nState := 210;
			ELSIF ipMoverApplication[nMoverIndex].std.P_MoveOnTrack.Error THEN
				   nErrorID := ipMoverApplication[nMoverIndex].std.P_MoveOnTrack.ErrorID;
				  nObjectID := ipMoverApplication[nMoverIndex].std.P_MoveOnTrack.stInfo.nObjectID;
				nObjectType := ipMoverApplication[nMoverIndex].std.P_MoveOnTrack.stInfo.nObjectType;
			END_IF		
		
		
	210: 	// do process
			Timer01(IN:=TRUE, PT:=T#1S);
			IF Timer01.Q THEN
				Timer01(IN:=FALSE);	
						
				IF nStationIndex = 1 THEN	
					// Station 1 toggeling mover destination to Station2 or Station3
					IF bToggleSwitch THEN
						ipMoverApplication[nMoverIndex].ProductData.nDestinationProcess := 2;
					ELSE
						ipMoverApplication[nMoverIndex].ProductData.nDestinationProcess := 3;		
					END_IF
					bToggleSwitch := NOT bToggleSwitch;					
				ELSE
					ipMoverApplication[nMoverIndex].ProductData.nDestinationProcess := 1;
				END_IF	
				
				nState := 220;
			END_IF

		
	220: 	// Send mover to the next station
			fMoverPosition     := fSendAwayPosition;	
			nTrackIndex        := nStationTrackIndex;		
			fMoverVelocity     :=    300.0;
			fMoverAcceleration :=  1_000.0;
			fMoverJerk         := 10_000.0;	
	
			stMoveParameters.direction := Tc3_Mc3PlanarMotion.MC_DIRECTION.mcDirectionPositive;
			stMoveParameters.gap       := 240.0;
			
			strInfo := CONCAT('Station: ', UINT_TO_STRING(nStationIndex));
			strInfo := CONCAT(strInfo, ' move to next Station:' );
			strInfo := CONCAT(strInfo, UINT_TO_STRING(nNextStationIndex));

			
			IF ipMoverApplication[nMoverIndex].std.P_MoveOnTrack.Done THEN

				FOR idx:=10 TO 1 BY -1 DO 
					strInfoHistory[idx] := strInfoHistory[idx-1];
				END_FOR
				strInfoHistory[0] := strInfo;		
			
				ipMoverApplication[nMoverIndex].std.MoveOnTrack( strInfo,
																 ipTrack[nTrackIndex].std,
																 fMoverPosition,
																 fMoverVelocity,
																 fMoverAcceleration,
																 fMoverJerk,
																 stMoveParameters.gap,
																 stMoveParameters.direction);
				nState := nState +1;
			END_IF		
		
		
	221: 	IF ipMoverApplication[nMoverIndex].std.P_MoveOnTrack.Active
			OR ipMoverApplication[nMoverIndex].std.P_MoveOnTrack.Done 
			THEN
				nState := 230;
			ELSIF ipMoverApplication[nMoverIndex].std.P_MoveOnTrack.Error THEN
				
				   nErrorID := ipMoverApplication[nMoverIndex].std.P_MoveOnTrack.ErrorID;
				  nObjectID := ipMoverApplication[nMoverIndex].std.P_MoveOnTrack.stInfo.nObjectID;
				nObjectType := ipMoverApplication[nMoverIndex].std.P_MoveOnTrack.stInfo.nObjectType;
			END_IF		
		
			
	230: 	// Mover to the list of the next station
			ipStation[nNextStationIndex].P_List.AddMover(P_List.RemoveFirstInList());
			nState := 500;	
	
		
	500: 	// Done for this cycle
			nState := 100;

END_CASE
END_METHOD

END_FUNCTION_BLOCK

// ---- 2_Application/Station/FB_Station_04_SW_Separate.TcPOU
FUNCTION_BLOCK FB_Station_04_SW_Separate EXTENDS FB_StationBase
VAR_INPUT
END_VAR
VAR_OUTPUT
END_VAR

METHOD ClearList : BOOL
VAR_INPUT
END_VAR
SUPER^.ClearList();
// Add aditional Data to Clear in Reset
// List and State will be cleared in master class
ClearList := TRUE;
END_METHOD

METHOD Processing : BOOL
VAR_INPUT
	i_nMachineState 	: INT;		// 1=starting, 2=Running
END_VAR


VAR_INST



	nMoverIndex						: UINT;
	fPositionOnTrack				: LREAL;
	nCurrentTrackIndex				: UDINT;
	fStationPositionOnTrack			: LREAL;
	nStationIndex					: UINT;
	
	nTrackNextStationPositionB		: UINT;
	nTrackNextStationPositionC		: UINT;	
	nNextStationIndexOutputB		: UINT;
	nNextStationIndexOutputC		: UINT;
	nTrackIndexOutputB				: UINT;
	nTrackIndexOutputC				: UINT;
	fSendAwayPositionOutputB		: LREAL;
	fSendAwayPositionOutputC		: LREAL;
	nNextStationIndex				: UINT;
	bSendToOutputB					: BOOL;
	bSendToOutputC					: BOOL;	
	fOutOfRangePosition				: LREAL;
	fMoverSpace						: LREAL;
	
	ClearTrig						: R_TRIG;
		
	nTrackindex						: UINT;
	fMoverPosition					: LREAL;
	fMoverVelocity					: LREAL;
	fMoverAcceleration				: LREAL;
	fMoverJerk						: LREAL;
	strInfo							: STRING;
	
	nErrorId						: UDINT;
	nObjectID						: UDINT;
	nObjectType						: UDINT;	
	
	nDestinationProcess				: UINT;
	nIncommingTrackOID				: UDINT;
			 
END_VAR

// Station - Switch-Seperate


ClearTrig(CLK:=bClearStation);
IF ClearTrig.Q THEN
	nState := 10;	
END_IF

CASE nState OF
	

	0:	// Waiting for initialization
		nState := 10;


	10:	// Init Station Parameters
				   nStationIndex := 4;		
		nNextStationIndexOutputB := 3;		
			  nTrackIndexOutputB := 3;		
		nNextStationIndexOutputC := 2;	
			  nTrackIndexOutputC := 2;	
			    	 fMoverSpace := 155 + 5.0;		
	    fSendAwayPositionOutputB := ipTrack[nTrackIndexOutputB].P_TrackLength/2 - fMoverSpace;		
		fSendAwayPositionOutputC := ipTrack[nTrackIndexOutputB].P_TrackLength/2 - fMoverSpace;		
			
		bClearStation := FALSE;
			   nState := 11;
	
	11: // Fail-safe check, just to make sure all variables have been assigned after doing copy&paste from the template	
		IF             nStationIndex > 0
		AND nNextStationIndexOutputB > 0
		AND       nTrackIndexOutputB > 0
		AND nNextStationIndexOutputC > 0 
		AND       nTrackIndexOutputC > 0 
		AND              fMoverSpace > 0
		AND fSendAwayPositionOutputB > 0
		AND fSendAwayPositionOutputC > 0
		AND              fMoverSpace > 0
		THEN
			nState := 20;
		END_IF

		
	20:	// Calculating station x-y-position 
		PositionOnTrack.fPositionOnTrack := 0.0;
		PositionOnTrack.nTrackId		 := UINT_TO_INT(nTrackIndexOutputB);
		ipTrack[PositionOnTrack.nTrackId].std.GetMoverPositionAt(PositionOnTrack.fPositionOnTrack, StationPosition);
		VisuPosX := StationPosition.x;
		VisuPosY := StationPosition.y;
		nState := 100;

			
		100: // Waiting for Mover
			IF P_List.P_FirstInList <> 0 THEN
				nMoverIndex := P_List.P_FirstInList.P_Id;
				nState := 110;
			END_IF
	
	
	110: // Decide to which Station the mover has to travel to next.	
			nDestinationProcess := ipMoverApplication[nMoverIndex].ProductData.nDestinationProcess;	
			nIncommingTrackOID	:= ipMoverApplication[nMoverIndex].std.P_SetOnTrack.TrackOID;
			nTrackindex := 0;
						
			CASE nDestinationProcess OF
			0: // -> OutputB
				nNextStationIndex  := nNextStationIndexOutputB;
				fMoverPosition     := fSendAwayPositionOutputB;
				nTrackindex        := nTrackIndexOutputB;		
		
			2: // -> OutputC
				nNextStationIndex  := nNextStationIndexOutputC;
				fMoverPosition     := fSendAwayPositionOutputC;
				nTrackindex        := nTrackIndexOutputC;				
	
			3: // -> OutputB
				nNextStationIndex  := nNextStationIndexOutputB;
				fMoverPosition     := fSendAwayPositionOutputB;
				nTrackindex        := nTrackIndexOutputB;		
			END_CASE
			
			IF nTrackindex > 0 THEN
				nState := 200;	
			END_IF


		

	200: 	// Send mover to the next station
			fMoverVelocity     :=    300.0;
			fMoverAcceleration :=  1_000.0;
			fMoverJerk         := 10_000.0;	
	
			stMoveParameters.direction := Tc3_Mc3PlanarMotion.MC_DIRECTION.mcDirectionPositive;
			stMoveParameters.gap       := 240.0;
		
			strInfo := CONCAT('Station: ', UINT_TO_STRING(nStationIndex));
			strInfo := CONCAT(strInfo, ' move to next Station:' );
			strInfo := CONCAT(strInfo, UINT_TO_STRING(nNextStationIndex));
		
	
			IF NOT ipMoverApplication[nMoverIndex].std.P_MoveOnTrack.Error THEN

				FOR idx:=10 TO 1 BY -1 DO 
					strInfoHistory[idx] := strInfoHistory[idx-1];
				END_FOR
				strInfoHistory[0] := strInfo;

		
				ipMoverApplication[nMoverIndex].std.MoveOnTrack( strInfo,
																 ipTrack[nTrackindex].std,
																 fMoverPosition,
																 fMoverVelocity,
																 fMoverAcceleration,
																 fMoverJerk,
																 stMoveParameters.gap,
																 stMoveParameters.direction);
																 																			 
		   		 nState := nState +1;
				 
			ELSIF ipMoverApplication[nMoverIndex].std.P_MoveOnTrack.Error THEN
				   nErrorID := ipMoverApplication[nMoverIndex].std.P_MoveOnTrack.ErrorID;
				  nObjectID := ipMoverApplication[nMoverIndex].std.P_MoveOnTrack.stInfo.nObjectID;
				nObjectType := ipMoverApplication[nMoverIndex].std.P_MoveOnTrack.stInfo.nObjectType;				
			END_IF
		

			
	201: 	IF ipMoverApplication[nMoverIndex].std.P_MoveOnTrack.Active
			OR ipMoverApplication[nMoverIndex].std.P_MoveOnTrack.Done 
			THEN
				nState := 210;
				
			ELSIF ipMoverApplication[nMoverIndex].std.P_MoveOnTrack.Error THEN
				
				   nErrorID := ipMoverApplication[nMoverIndex].std.P_MoveOnTrack.ErrorID;
				  nObjectID := ipMoverApplication[nMoverIndex].std.P_MoveOnTrack.stInfo.nObjectID;
				nObjectType := ipMoverApplication[nMoverIndex].std.P_MoveOnTrack.stInfo.nObjectType;
			END_IF			
	

	210: // Check if Mover passed the junction point		
			IF ipMoverApplication[nMoverIndex].std.P_SetOnTrack.TrackOID <> nIncommingTrackOID THEN 
				nState := 220;
			END_IF

	
	220: // Mover to the list of the next station
		ipStation[nNextStationIndex].P_List.AddMover(P_List.RemoveFirstInList());
		nState := 500;	
	
		
	500: // done for this cycle
		nState := 100;

END_CASE
END_METHOD

END_FUNCTION_BLOCK

// ---- 2_Application/Station/FB_Station_05_SW_Merge.TcPOU
FUNCTION_BLOCK FB_Station_05_SW_Merge EXTENDS FB_StationBase
VAR_INPUT
END_VAR
VAR_OUTPUT
END_VAR

METHOD ClearList : BOOL
VAR_INPUT
END_VAR
SUPER^.ClearList();
// Add aditional Data to Clear in Reset
// List and State will be cleared in master class
ClearList := TRUE;
END_METHOD

METHOD Processing : BOOL
VAR_INPUT
	i_nMachineState 	: INT;		// 1=Starting, 2=Running
END_VAR

VAR_INST
	
	ClearTrig					: R_TRIG;
	
	fStationPositionOnTrack		: LREAL;

	nStationIndex				: UINT;
	nNextStationIndex			: UINT;
	nNextStationTrackIndex		: UINT;
	nMoverIndex					: UINT;
	nNextStationIndexOutputA	: UINT;
	nTrackIndexOutputA			: UINT;	
	fSendAwayPositionOutputA	: LREAL;	

	nMoverIndexInputB			: UINT;
	nMoverIndexInputC			: UINT;
	nTrackIndex					: UINT;
	fMoverPosition				: LREAL;
	fMoverVelocity				: LREAL;
	fMoverAcceleration			: LREAL;
	fMoverJerk					: LREAL;
	nIncommingTrackOID			: UDINT;
	
	nErrorId					: UDINT;
	nObjectID					: UDINT;
	nObjectType					: UDINT;	
	
END_VAR

// Station - Switch-Merge	


ClearTrig(CLK:=bClearStation);
IF ClearTrig.Q THEN
	nState := 10;	
END_IF

CASE nState OF
	
	0:	// Waiting for initialization
		nState := 10;
	

	
	10:	// Init Station-Parameters	
					   nStationIndex := 5;		
			nNextStationIndexOutputA := 1;	
				  nTrackIndexOutputA := 1;		
			fSendAwayPositionOutputA := 240.0;			
				
			bClearStation := FALSE;
			       nState := 11;

	11: // Fail-safe check, just to make sure all variables have been assigned after doing copy&paste from the template
		IF             nStationIndex > 0
		AND nNextStationIndexOutputA > 0
		AND       nTrackIndexOutputA > 0
		AND fSendAwayPositionOutputA > 0 
		THEN
			nState := 20;
		END_IF

		
	20:	// Calculating station x-y-position 
		PositionOnTrack.fPositionOnTrack := 0.0;
		PositionOnTrack.nTrackId		 := UINT_TO_INT(nTrackIndexOutputA);
		ipTrack[PositionOnTrack.nTrackId].std.GetMoverPositionAt(PositionOnTrack.fPositionOnTrack, StationPosition);
		VisuPosX := StationPosition.x;
		VisuPosY := StationPosition.y;
		nState := 100;
			   
		
	100: // Waiting for Mover on Input_B or Input_C
		IF P_List.P_FirstInList = 0 THEN
			nMoverIndexInputB := 0;
			nMoverIndexInputC := 0;
		
			IF P_List_Input_B.P_FirstInList <> 0 THEN
				nMoverIndexInputB := P_List_Input_B.P_FirstInList.P_Id;
			END_IF		
			
			IF P_List_Input_C.P_FirstInList <> 0 THEN
				nMoverIndexInputC := P_List_Input_C.P_FirstInList.P_Id;
			END_IF				
			
			IF nMoverIndexInputB > 0 
			OR nMoverIndexInputC > 0
			THEN
				 nState := 110;
			END_IF
		ELSE
			nState := 120;
		END_IF
		
		
	110: // Priority: B comes first  
		IF nMoverIndexInputB > 0 THEN
			P_List.AddMover(P_List_Input_B.RemoveFirstInList());
		ELSE
			P_List.AddMover(P_List_Input_C.RemoveFirstInList());
		END_IF	
		nState := 120;
		
		
	120: // Processing mover to next Station
		IF P_List.P_FirstInList <> 0 THEN
			       nMoverIndex := P_List.P_FirstInList.P_Id;
			nIncommingTrackOID := ipMoverApplication[nMoverIndex].std.P_SetOnTrack.TrackOID;
			            nState := 200;
		END_IF
		
			 
	200: 	// Send mover to the next station output A
			nNextStationIndex  := nNextStationIndexOutputA;
			nTrackIndex 	   := nTrackIndexOutputA;			
			fMoverPosition     := fSendAwayPositionOutputA;
			fMoverVelocity     :=    300.0;
			fMoverAcceleration :=  1_000.0;
			fMoverJerk         := 10_000.0;	
	
			stMoveParameters.direction := Tc3_Mc3PlanarMotion.MC_DIRECTION.mcDirectionPositive;
			stMoveParameters.gap       := 240.0;
		
			strInfo := CONCAT('Station: ', UINT_TO_STRING(nStationIndex));
			strInfo := CONCAT(strInfo, ' move to next Station:' );
			strInfo := CONCAT(strInfo, UINT_TO_STRING(nNextStationIndex));
			

			
	
			IF NOT ipMoverApplication[nMoverIndex].std.P_MoveOnTrack.Error THEN

				FOR idx:=10 TO 1 BY -1 DO 
					strInfoHistory[idx] := strInfoHistory[idx-1];
				END_FOR
				strInfoHistory[0] := strInfo;				

				ipMoverApplication[nMoverIndex].std.MoveOnTrack( strInfo,
																 ipTrack[nTrackIndex].std,
																 fMoverPosition,
																 fMoverVelocity,
																 fMoverAcceleration,
																 fMoverJerk,
																 stMoveParameters.gap,
																 stMoveParameters.direction);
																 
																 
			ipMoverApplication[nMoverIndex].P_nTrackId := nNextStationTrackIndex;
															 
		    nState := nState +1;
			
			ELSIF ipMoverApplication[nMoverIndex].std.P_MoveOnTrack.Error THEN
				   nErrorID := ipMoverApplication[nMoverIndex].std.P_MoveOnTrack.ErrorID;
				  nObjectID := ipMoverApplication[nMoverIndex].std.P_MoveOnTrack.stInfo.nObjectID;
				nObjectType := ipMoverApplication[nMoverIndex].std.P_MoveOnTrack.stInfo.nObjectType;				
			END_IF			
			

	201: 	IF ipMoverApplication[nMoverIndex].std.P_MoveOnTrack.Error THEN
				   nErrorID := ipMoverApplication[nMoverIndex].std.P_MoveOnTrack.ErrorID;
				  nObjectID := ipMoverApplication[nMoverIndex].std.P_MoveOnTrack.stInfo.nObjectID;
				nObjectType := ipMoverApplication[nMoverIndex].std.P_MoveOnTrack.stInfo.nObjectType;		
			ELSE
				IF ipMoverApplication[nMoverIndex].std.P_MoveOnTrack.Active 
				OR ipMoverApplication[nMoverIndex].std.P_MoveOnTrack.Done
				THEN
					nState := 210;
				END_IF
			END_IF

			
	210: // Check if Mover passed the junction point		
		IF ipMoverApplication[nMoverIndex].std.P_SetOnTrack.TrackOID <> nIncommingTrackOID THEN 
			nState := 220;
		END_IF
	
	
	220: // Check if Mover is out of range
		IF ipMoverApplication[nMoverIndex].std.P_SetOnTrack.SetPos > 120.0 THEN 
			nState := 230;
		END_IF

	
	230: // Mover to the list of the next station
		ipStation[nNextStationIndex].P_List.AddMover(P_List.RemoveFirstInList());
		nState := 500;	
	
		
	500: // done for this cycle
		nState := 100;
		
	
END_CASE
END_METHOD

END_FUNCTION_BLOCK

// ---- 1_Industry/FB_SK_StateManager.TcPOU
FUNCTION_BLOCK FB_SK_StateManager

VAR
	bStartUpDone		: BOOL;	
	bFirstAbortDone		: BOOL;
	
	eCommand			: E_XMotion_Command;	
	eCommandOld			: E_XMotion_Command;
	eStatus				: E_XMotion_Status;	
	nCommandCounter		: UDINT;

END_VAR

METHOD PUBLIC Cycle
VAR_INPUT
END_VAR


	IF NOT bStartUpDone THEN					
		eStatus := E_XMotion_Status.StartUp;
	ELSIF NOT bFirstAbortDone THEN
		eStatus := E_XMotion_Status.Aborting;
	ELSE

		IF eCommand <> eCommandOld THEN
			eCommandOld := eCommand;
	
			nCommandCounter := nCommandCounter +1;
			
			
			CASE eCommand OF
				
			
			E_XMotion_Command.Abort:	
						eStatus := E_XMotion_Status.Aborting;	
			
			E_XMotion_Command.Reset:
						IF eStatus = E_XMotion_Status.Aborted THEN
							eStatus := E_XMotion_Status.Resetting;	
						END_IF
				
			E_XMotion_Command.Prepare:
						IF eStatus = E_XMotion_Status.Stopped THEN
							eStatus := E_XMotion_Status.Preparing;	
						END_IF	
			
			E_XMotion_Command.Start:
						IF eStatus = E_XMotion_Status.Prepared THEN
							eStatus := E_XMotion_Status.Execute;	
						END_IF	

			E_XMotion_Command.HoldOnError:
						eStatus := E_XMotion_Status.HoldOnError;

					
			END_CASE
		END_IF
		
	END_IF
END_METHOD

METHOD PUBLIC StateComplete : BOOL
VAR_INPUT
END_VAR




	CASE eStatus OF
		
	E_XMotion_Status.StartUp:
				bStartUpDone := TRUE;
				
	E_XMotion_Status.Aborting:
				bFirstAbortDone := TRUE;	
				eStatus := E_XMotion_Status.Aborted;	
	
	E_XMotion_Status.Resetting:
				eStatus := E_XMotion_Status.Stopped;
		
	E_XMotion_Status.Preparing:
				eStatus := E_XMotion_Status.Prepared;
	
				
	END_CASE
END_METHOD

PROPERTY Status : E_XMotion_Status
GET
Status := eStatus;
END_GET
END_PROPERTY

PROPERTY XMotionCommand : E_XMotion_Command
SET
eCommand := XMotionCommand;
END_SET
END_PROPERTY

END_FUNCTION_BLOCK

// ---- 1_Industry/FB_OperationalControl.TcPOU
FUNCTION_BLOCK FB_OperationalControl
VAR_INPUT

	bStartCommand 		: BOOL;
	bStopCommand 		: BOOL;		
	bQuitCommand 		: BOOL;
	bExceptionCommand	: BOOL;

END_VAR
VAR_OUTPUT
	bStartLamp 			: BOOL;
	bStopLamp 			: BOOL;
	bQuitLamp 			: BOOL;
	bEStopLamp			: BOOL;
	bStopping			: BOOL;
	bStopped			: BOOL;
	bStarting 			: BOOL;
	bRunning			: BOOL;
	sResult 			: STRING;
	nResult				: INT;
END_VAR

VAR_IN_OUT
	XTags		: ST_XTags;
END_VAR

VAR
	nMachineState		: INT;
	bStartUpFlag		: BOOL;
	bStartUpDone		: BOOL;
	bError				: BOOL;
	bStartSequence		: BOOL;
	bStopSequence		: BOOL;
	bStartLampBlink		: BOOL;
	bStopLampBlink		: BOOL;
	nErrorSequence		: INT;
	tBlinker			: TON;
	bBlinker			: BOOL;

	bCheckCurrentMachineState	: BOOL;

	nProcessFeedback		: UDINT;

	rtMoverErrordetection	: R_TRIG;
	bMoverErrorDetected		: BOOL;
	
END_VAR


	helper();

	
	// Check for system start-up
	IF NOT bStartUpDone THEN
		IF XTags.Status = E_XMotion_Status.StartUp THEN
			bStartUpFlag := TRUE;
		END_IF			
		IF bStartUpFlag AND XTags.Status = E_XMotion_Status.Aborted THEN	
			IF NOT bStartUpDone THEN
				bStartUpDone   := TRUE;
			    bStartSequence := FALSE;
		        bStopSequence  := TRUE;
			END_IF
		END_IF	
		sResult := 'Machine Start-Up';
	END_IF
	

	// Check start signal
	IF bStartCommand 
	AND NOT bStopCommand 
	AND NOT bExceptionCommand
	AND NOT bStopSequence
	AND NOT bError
	THEN 
		bStartSequence := TRUE;
		bStopSequence  := FALSE;
	END_IF
	
	// Check stop signal
	IF bStopCommand 
	AND NOT bExceptionCommand
	AND NOT bError
	THEN
		bStartSequence := FALSE;
		bStopSequence  := TRUE;
	END_IF 
	
		
	ErrorSequence();
	StartSequence();
	StopSequence();
	SyncSequence();

ACTION ErrorSequence:





	
CASE nErrorSequence OF
		
	0:	// Checking mover error  
		IF ipMotionSystemApplication <> 0 THEN
			rtMoverErrordetection(CLK:=ipMotionSystemApplication.P_bMoverError);
			IF rtMoverErrordetection.Q THEN
				bMoverErrorDetected := TRUE;
			END_IF
		END_IF	
		
		// In case of an exception e.g. E-Stop, start the error sequence
		IF bExceptionCommand THEN    // -> Exception from extern e.g. E-Stop Button
			XTags.Command := E_XMotion_Command.Abort;
			nErrorSequence := 5;
		ELSE
			IF bMoverErrorDetected THEN	// -> Exception from a Mover e.g. FollowingError
				XTags.Command := E_XMotion_Command.HoldOnError;
				nErrorSequence := 5;
			END_IF			
		END_IF	

		
	5:	// In case of an exception e.g. E-Stop, start the error sequence
		 bStartSequence := FALSE;
		 bStopSequence  := FALSE;
			 bStartLamp := FALSE;
			  bStopLamp := FALSE;
			  bQuitLamp := FALSE;
		bStartLampBlink := FALSE;
		 bStopLampBlink := FALSE;	 
				 bError := TRUE;	
		
	     nErrorSequence := 10;
		
	
	10:	// Waiting till the event is gone e.g. E-Stop has been pulled out.		
		bEStopLamp := bBlinker;
		sResult := 'Error pending';	
		IF NOT bExceptionCommand THEN
			    bEStopLamp := FALSE;
			nErrorSequence := 20;
		END_IF
			
		
	20:	// Wait for error-quit	
		bQuitLamp := bBlinker;
		
		IF ipMotionSystemApplication.P_bMoverError THEN
			sResult := 'Mover Error / Waiting for error-quit';
		ELSE
			sResult := 'Waiting for error-quit';
		END_IF

		IF bExceptionCommand THEN
			nErrorSequence := 5;
		ELSIF bQuitCommand THEN
			bMoverErrorDetected := FALSE;
			     nErrorSequence := 30;
		END_IF
		
		
	30: // Sending abort-command to the StarterKit-StateMachine.
		XTags.Command := E_XMotion_Command.Abort;
		     bQuitLamp := bBlinker;
		       sResult := 'Error-Quit - sending abort-command';		
		nErrorSequence := 40;
		
	  
	40: // Waiting for StarterKit-StateMachine in state Aborted.
		IF XTags.Status = E_XMotion_Status.Aborted THEN
			bQuitLamp := FALSE;
		    bStopLamp := TRUE;
			   bError := FALSE;
			  sResult := 'Error-Quit successful';	
			  
			nErrorSequence := 0;
		END_IF		  

	END_CASE
END_ACTION

ACTION helper:




	IF bStartLampBlink THEN
		bStartLamp := bBlinker;
	END_IF
	
	IF bStopLampBlink THEN
		bStopLamp := bBlinker;
	END_IF
	

	tBlinker(IN:=TRUE, PT:=T#500MS);
	IF tBlinker.Q THEN
		bBlinker := NOT bBlinker;
		tBlinker(IN:=FALSE);
	END_IF
END_ACTION

PROPERTY P_nProcessFeedback : UDINT
SET
nProcessFeedback := P_nProcessFeedback;
END_SET
END_PROPERTY

ACTION StartSequence:


	
	
	
	// Start-Sequence, will run in case of start-signal 
	IF bStartSequence THEN
		CASE XTags.Status OF
			
			E_XMotion_Status.StartUp:	// Do nothing
										bStartSequence := FALSE;
										sResult := 'Impossible - Machine is still in Start-Up procedure';	
										
			E_XMotion_Status.Aborting:	// Do nothing
										bStartSequence := FALSE;
										sResult := 'Impossible - Machine is in Aborting sequence';	
		
			E_XMotion_Status.Aborted:	// Reset-Command brings you to the next stage
										  nMachineState := 1;
										bStartLampBlink := TRUE;
										      bStopLamp := FALSE;
										  XTags.Command := E_XMotion_Command.Reset;
										sResult := 'Starting - command reset issued';
		
			E_XMotion_Status.Resetting: // Wait for next stage
			  						      nMachineState := 1;
										bStartLampBlink := TRUE;
										      bStopLamp := FALSE;
										sResult := 'Starting - Machine is resetting';
										
			E_XMotion_Status.Stopped:	// Prepare-Command brings you to the next stage
									      nMachineState := 2;
										bStartLampBlink := TRUE;
										  XTags.Command := E_XMotion_Command.Prepare;
										sResult := 'Starting - command prepare issued';	
		
			E_XMotion_Status.Preparing: // Wait for next stage
										  nMachineState := 3;
										bStartLampBlink := TRUE;
										      bStopLamp := FALSE;
										sResult := 'Starting - Machine is preparing';
		
			E_XMotion_Status.Prepared:	// Start-Command brings you to the next stage
										  nMachineState := 3;
										bStartLampBlink := TRUE;
										      bStopLamp := FALSE;
										  XTags.Command := E_XMotion_Command.Start;
										sResult := 'Starting - command start issued';	 
		
			E_XMotion_Status.Execute:	// System is running
										 nMachineState := 4;
									   bStartLampBlink := FALSE;
											 bStopLamp := FALSE;
										    bStartLamp := TRUE;
										bStartSequence := FALSE;
										sResult := 'Machine is running';
		
		END_CASE
	END_IF
END_ACTION

ACTION StopSequence:





	

	// Stop-Sequence, will run in case of stop-signal 
	IF bStopSequence THEN
		     bStartLamp := FALSE;
		bStartLampBlink := FALSE;
		
		CASE XTags.Status OF
			
			E_XMotion_Status.StartUp:	// Do nothing
										bStopSequence := FALSE;
										sResult := 'Impossible - Machine is still in Start-Up procedure';	
										
			E_XMotion_Status.Aborting:	// Do nothing
										sResult := 'Impossible - Machine is in Aborting sequence';	
		
			E_XMotion_Status.Aborted:	// System is stopped
										 nMachineState := 2;
			                            bStopLampBlink := FALSE;
			                                 bStopLamp := TRUE;
										 bStopSequence := FALSE;
										sResult := 'Machine is stopped';
		
			E_XMotion_Status.Resetting: // Sending abort-command
										 nMachineState := 1;
										bStopLampBlink := TRUE;
										 XTags.Command := E_XMotion_Command.Abort;
										sResult := 'Machine is resetting - sending abort-command';
										
			E_XMotion_Status.Stopped:	// Sending abort-command
										 nMachineState := 1;
										bStopLampBlink := TRUE;
										 XTags.Command := E_XMotion_Command.Abort;
										sResult := 'Machine is stopped - sending abort-command';
		
			E_XMotion_Status.Preparing: // Sending abort-command
										 nMachineState := 1;
										 nMachineState := 1;
										bStopLampBlink := TRUE;
										 XTags.Command := E_XMotion_Command.Abort;
										sResult := 'Machine is preparing - sending abort-command';
		
			E_XMotion_Status.Prepared:	// Sending abort-command
										 nMachineState := 1;
										bStopLampBlink := TRUE;
										 XTags.Command := E_XMotion_Command.Abort;
										sResult := 'Machine is prepared - sending abort-command';
		
			E_XMotion_Status.Execute:	// Sending abort-command
									     nMachineState := 1;
										bStopLampBlink := TRUE;
										    bStartLamp := FALSE;
										 XTags.Command := E_XMotion_Command.Abort;
										sResult := 'Machine is executing - sending abort-command';
		
		END_CASE

	END_IF
END_ACTION

ACTION SyncSequence:




	

	CASE nMachineState OF
		
	0:	// Machine state = undefined
		bStopping := FALSE;
		bStopped  := FALSE;
		bStarting := FALSE;
		bRunning  := FALSE;	
				
	1:	// Machine state = stopping	
		bStopping := TRUE;
		bStopped  := FALSE;
		bStarting := FALSE;
		bRunning  := FALSE;	
		IF XTags.Status <> E_XMotion_Status.Aborting THEN
			bCheckCurrentMachineState := TRUE;
		END_IF
		
	2:	// Machine state = stopped	
		bStopping := FALSE;
		bStopped  := TRUE;
		bStarting := FALSE;
		bRunning  := FALSE;	
		IF XTags.Status <> E_XMotion_Status.Stopped THEN
			bCheckCurrentMachineState := TRUE;
		END_IF
	
	3:	// Machine state = starting	
		bStopping := FALSE;
		bStopped  := FALSE;
		bStarting := TRUE;
		bRunning  := FALSE;
		IF XTags.Status <> E_XMotion_Status.Preparing THEN
			bCheckCurrentMachineState := TRUE;
		END_IF					
		
	4:	// Machine state = running	
		bStopping := FALSE;
		bStopped  := FALSE;
		bStarting := FALSE;
		bRunning  := TRUE;		
		IF XTags.Status <> E_XMotion_Status.Execute THEN
			bCheckCurrentMachineState := TRUE;
		END_IF
		
	END_CASE



	// Syncronizing with StarterKit-StateMachine
	IF bCheckCurrentMachineState 
	AND NOT bError
	THEN
		bCheckCurrentMachineState := FALSE;
		
		CASE XTags.Status OF
			
			E_XMotion_Status.StartUp:	// Do nothing
										sResult := 'Machine Start-Up';
										
										bStartSequence := FALSE;
										 bStopSequence := FALSE;
										 nMachineState := 0;
											
										
			E_XMotion_Status.Aborting:	// Do nothing
										        sResult := 'Machine Aborting';	
										  nMachineState := 1;
										bStartLampBlink := FALSE;
										     bStartLamp := FALSE;
										 bStopLampBlink := TRUE;
										      bStopLamp := FALSE;
		
			E_XMotion_Status.Aborted:	// Reset-Command brings you to the next stage
										        sResult := 'Machine Aborted';	
										  nMachineState := 2;
										bStartLampBlink := FALSE;
										     bStartLamp := FALSE;
										 bStopLampBlink := FALSE;
										      bStopLamp := TRUE;

		
			E_XMotion_Status.Resetting: // Wait for next stage
										        sResult := 'Machine Resetting';	
			  						      nMachineState := 1;
										bStartLampBlink := TRUE;
										      bStopLamp := FALSE;

										
			E_XMotion_Status.Stopped:	// Prepare-Command brings you to the next stage
									   	        sResult := 'Stopped';
									      nMachineState := 2;
	
		
			E_XMotion_Status.Preparing: // Wait for next stage
												sResult := 'Machine Preparing';
										  nMachineState := 3;
										bStartLampBlink := TRUE;
										      bStopLamp := FALSE;

		
			E_XMotion_Status.Prepared:	// Start-Command brings you to the next stage
										        sResult := 'Prepared';
										  nMachineState := 3;
										bStartLampBlink := TRUE;
										      bStopLamp := FALSE;
	 
		
			E_XMotion_Status.Execute:	// System is running
									           sResult := 'Machine is Running';
										 nMachineState := 4;
									   bStartLampBlink := FALSE;
											 bStopLamp := FALSE;
										    bStartLamp := TRUE;
										bStartSequence := FALSE;
		
		END_CASE
	END_IF
END_ACTION

END_FUNCTION_BLOCK

// ---- 1_Industry/FB_VisStarterKitStateMachine.TcPOU
FUNCTION_BLOCK FB_VisStarterKitStateMachine

VAR_IN_OUT

	iq_stVisControl  : ST_VisControl;
	iq_XTags		 : ST_XTags;
		
END_VAR


VAR
		
	diStatusOld : DINT := -1;
	
	
	// Operator-Control-Pad 
	bOCStartButton			: BOOL;
	bOCStopButton			: BOOL;
	bOCQuitButton			: BOOL;
	bOCEStopButton			: BOOL;
	
	bOCStopLamp				: BOOL;
	bOCStartLamp			: BOOL;
	bOCQuitLamp				: BOOL;
	bOCEStopLamp			: BOOL;
	
	bOCMessageColorGreen	: BOOL;
	bOCMessageColorRed		: BOOL;	
	
	sOCResultText			: STRING;
	sDisplayText			: STRING;
	nStringPosition			: INT;
	nStringLength			: INT;
	nDisplayLenght			: INT := 28;
		
	nOCResultNumber			: INT;
	DisplayTimer			: TON;
	
	rtNoCommandTrigger		: R_TRIG;
	
	bInitScreenDone			: BOOL;
	nVisArrangement			: INT;
	nVisArrangementMem		: INT;
	nVisArrangementSet		: INT;
	
END_VAR




	ScreenArrangement();
	
	StarterKitStateMachine();

	OperatorInterface();

PROPERTY PUBLIC bOCEStopButtonState : BOOL
GET
bOCEStopButtonState := bOCEStopButton;
END_GET
END_PROPERTY

PROPERTY PUBLIC bOCEStopLampState : BOOL
SET
bOCEStopLamp := bOCEStopLampState;
END_SET
END_PROPERTY

PROPERTY PUBLIC bOCQuitButtonState : BOOL
GET
bOCQuitButtonState := bOCQuitButton;
END_GET
END_PROPERTY

PROPERTY PUBLIC bOCQuitLampState : BOOL
SET
bOCQuitLamp := bOCQuitLampState;
END_SET
END_PROPERTY

PROPERTY PUBLIC bOCStartButtonState : BOOL
GET
bOCStartButtonState := bOCStartButton;
END_GET
END_PROPERTY

PROPERTY PUBLIC bOCStartLampState : BOOL
SET
bOCStartLamp := bOCStartLampState;
END_SET
END_PROPERTY

PROPERTY PUBLIC bOCStopButtonState : BOOL
GET
bOCStopButtonState := bOCStopButton;
END_GET
END_PROPERTY

PROPERTY PUBLIC bOCStopLampState : BOOL
SET
bOCStopLamp := bOCStopLampState;
END_SET
END_PROPERTY

PROPERTY PUBLIC nOCResult : int
SET
nOCResultNumber := nOCResult;
END_SET
END_PROPERTY

ACTION OperatorInterface:



	

		
		
		bOCStartButton 	:= iq_stVisControl.stOperatorPad.bStartButtunState;
		bOCStopButton  	:= iq_stVisControl.stOperatorPad.bStopButtonState; 
		bOCQuitButton	:= iq_stVisControl.stOperatorPad.bQuitButtonState;
		bOCEStopButton	:= iq_stVisControl.stOperatorPad.bEStopButtonState;
		
		
		iq_stVisControl.stOperatorPad.bStartButtonLamp 		:= bOCStartLamp;
		iq_stVisControl.stOperatorPad.bStopButtonLamp  		:= bOCStopLamp;
		iq_stVisControl.stOperatorPad.bQuitButtonLamp  		:= bOCQuitLamp;
		iq_stVisControl.stOperatorPad.bEStopButtonLamp 		:= bOCEStopLamp;
		iq_stVisControl.stOperatorPad.bMessageColorGreen 	:= bOCMessageColorGreen;
		iq_stVisControl.stOperatorPad.bMessageColorRed   	:= bOCMessageColorRed;
		
			
		nStringLength := LEN(sOCResultText);	
		IF nStringLength > nDisplayLenght THEN
			sDisplayText := MID(sOCResultText,nDisplayLenght,nStringPosition);
		
			DisplayTimer(IN:=TRUE, PT:=T#500MS);
			IF DisplayTimer.Q THEN
				DisplayTimer(IN:=FALSE);
				nStringPosition := nStringPosition +1;
				
				IF nStringPosition > (nStringLength - nDisplayLenght) THEN
					nStringPosition := 1;
				END_IF
			END_IF
		ELSE
			sDisplayText := sOCResultText;
		END_IF
		iq_stVisControl.stOperatorPad.sMessage := sDisplayText;
END_ACTION

ACTION ScreenArrangement:






	// Decide which Pad shall be shown at system boot:
	IF NOT bInitScreenDone THEN
		bInitScreenDone := TRUE;

		iq_stVisControl.stControlPad.bVisInvisibleButton  := FALSE;		
		iq_stVisControl.stOperatorPad.bVisInvisibleButton := FALSE;
	END_IF


	// Check which Pad shall be shown right now:
	IF iq_stVisControl.stControlPad.bVisInvisibleButton THEN
		iq_stVisControl.stControlPad.bVisInvisible := TRUE;
	ELSE
		iq_stVisControl.stControlPad.bVisInvisible := FALSE;
	END_IF	

	IF iq_stVisControl.stOperatorPad.bVisInvisibleButton THEN
		iq_stVisControl.stOperatorPad.bVisInvisible := TRUE;
	ELSE
		iq_stVisControl.stOperatorPad.bVisInvisible := FALSE;
	END_IF		
	

	// Determine current visualisation arrangement:
	IF  iq_stVisControl.stControlPad.bVisInvisible 
	AND iq_stVisControl.stOperatorPad.bVisInvisible
	THEN
		nVisArrangement := 1;
		
	ELSIF ( NOT iq_stVisControl.stControlPad.bVisInvisible
			AND iq_stVisControl.stOperatorPad.bVisInvisible) 
	THEN
		nVisArrangement := 2;
		
	ELSIF ( NOT iq_stVisControl.stOperatorPad.bVisInvisible 
			AND iq_stVisControl.stControlPad.bVisInvisible )
	THEN
		nVisArrangement := 3;
	ELSIF (     NOT iq_stVisControl.stControlPad.bVisInvisible 
			AND NOT iq_stVisControl.stOperatorPad.bVisInvisible)
	THEN
		nVisArrangement := 4;
	END_IF
	
	
	
	// Arranging all frame positions according to current arrangement:
	IF nVisArrangement <> nVisArrangementMem THEN
		nVisArrangementMem := nVisArrangement;
		nVisArrangementSet := nVisArrangement;
	END_IF
		
	CASE nVisArrangementSet OF 	
	
	1:  nVisArrangementSet := 0;
		
		iq_stVisControl.stControlPad.nFramePositionX   :=  0;
		iq_stVisControl.stControlPad.nFramePositionY   :=  0;
		iq_stVisControl.stControlPad.nButtonPositionX  :=  0;
		iq_stVisControl.stControlPad.nButtonPositionY  := 55;
		
		iq_stVisControl.stOperatorPad.nFramePositionX  :=  0;
		iq_stVisControl.stOperatorPad.nFramePositionY  :=  0;
		iq_stVisControl.stOperatorPad.nButtonPositionX :=  0;
		iq_stVisControl.stOperatorPad.nButtonPositionY := 55;
				
	2: 	nVisArrangementSet := 0;
	
		iq_stVisControl.stControlPad.nFramePositionX   :=  0;
		iq_stVisControl.stControlPad.nFramePositionY   := 60;	
		iq_stVisControl.stOperatorPad.nButtonPositionX :=  0;
		iq_stVisControl.stOperatorPad.nButtonPositionY := 55;	
	
	3:	nVisArrangementSet := 0;
	
		iq_stVisControl.stControlPad.nButtonPositionX  :=  0;
		iq_stVisControl.stControlPad.nButtonPositionY  := -2;
		iq_stVisControl.stOperatorPad.nFramePositionX  :=  0;
		iq_stVisControl.stOperatorPad.nFramePositionY  :=  0;
	
	4:	nVisArrangementSet := 0;
	
		iq_stVisControl.stControlPad.nFramePositionX   :=  0;
		iq_stVisControl.stControlPad.nFramePositionY   :=  0;
		iq_stVisControl.stOperatorPad.nFramePositionX  :=  0;
		iq_stVisControl.stOperatorPad.nFramePositionY  :=  0;
	
	END_CASE
END_ACTION

PROPERTY PUBLIC sOCResultTextDisplay : STRING
SET
sOCResultText := sOCResultTextDisplay;
END_SET
END_PROPERTY

ACTION StarterKitStateMachine:


	// Setting XTag-Commands according to user-commands
	IF    iq_stVisControl.stControlPad.bButtonState_Abort THEN
				rtNoCommandTrigger(CLK:=FALSE);
				iq_XTags.Command  := E_XMotion_Command.Abort;	
	ELSIF iq_stVisControl.stControlPad.bButtonState_Reset THEN
				rtNoCommandTrigger(CLK:=FALSE);
				iq_XTags.Command  := E_XMotion_Command.Reset;	
	ELSIF iq_stVisControl.stControlPad.bButtonState_Prepare THEN
				rtNoCommandTrigger(CLK:=FALSE);
				iq_XTags.Command  := E_XMotion_Command.Prepare;	
	ELSIF iq_stVisControl.stControlPad.bButtonState_Start THEN
				rtNoCommandTrigger(CLK:=FALSE);
				iq_XTags.Command  := E_XMotion_Command.Start;	
	ELSE
			rtNoCommandTrigger(CLK:=TRUE);
			IF rtNoCommandTrigger.Q THEN
				iq_XTags.Command  := E_XMotion_Command.NoCommand;
			END_IF
	END_IF


	
	
	// Setting Vis display according to current status	
	iq_stVisControl.stControlPad.iAbortSequenceState   := iq_XTags.States.nAbortState;
	iq_stVisControl.stControlPad.iResetSequenceState   := iq_XTags.States.nResetState;
	iq_stVisControl.stControlPad.iPrepareSequenceState := iq_XTags.States.nPrepareState;
	iq_stVisControl.stControlPad.iStartSequenceState   := iq_XTags.States.nStartState;
	

	IF iq_XTags.Status <> diStatusOld THEN
		diStatusOld := iq_XTags.Status;	
	
		iq_stVisControl.stControlPad.bAbortSequenceStateInvisible 	:= TRUE;
		iq_stVisControl.stControlPad.bResetSequenceStateInvisible 	:= TRUE;
		iq_stVisControl.stControlPad.bPrepareSequenceStateInvisible := TRUE;
		iq_stVisControl.stControlPad.bStartSequenceStateInvisible	:= TRUE;
		
		iq_stVisControl.stControlPad.bStateSignalAbortBlue     := FALSE;
		iq_stVisControl.stControlPad.bStateSignalAbortYellow   := FALSE;
		iq_stVisControl.stControlPad.bStateSignalAbortGreen    := FALSE;
		iq_stVisControl.stControlPad.bStateSignalResetYellow   := FALSE;
		iq_stVisControl.stControlPad.bStateSignalResetGreen    := FALSE;		
		iq_stVisControl.stControlPad.bStateSignalResetYellow   := FALSE;
		iq_stVisControl.stControlPad.bStateSignalResetGreen    := FALSE;		
		iq_stVisControl.stControlPad.bStateSignalPrepareYellow := FALSE;
		iq_stVisControl.stControlPad.bStateSignalPrepareGreen  := FALSE;		
		iq_stVisControl.stControlPad.bStateSignalExecuteYellow := FALSE;
		iq_stVisControl.stControlPad.bStateSignalExecuteGreen  := FALSE;	

		IF 	   iq_XTags.Status = E_XMotion_Status.Aborting THEN
					iq_stVisControl.stControlPad.bAbortSequenceStateInvisible := FALSE;
					iq_stVisControl.stControlPad.bStateSignalAbortYellow   	  := TRUE;		
		ELSIF iq_XTags.Status = E_XMotion_Status.Aborted THEN
					iq_stVisControl.stControlPad.bStateSignalAbortGreen := TRUE;
		ELSIF iq_XTags.Status = E_XMotion_Status.Resetting THEN
					iq_stVisControl.stControlPad.bResetSequenceStateInvisible := FALSE;
					iq_stVisControl.stControlPad.bStateSignalResetYellow      := TRUE;
		ELSIF iq_XTags.Status = E_XMotion_Status.Stopped THEN
					iq_stVisControl.stControlPad.bStateSignalResetGreen := TRUE;
		ELSIF iq_XTags.Status = E_XMotion_Status.Preparing THEN
					iq_stVisControl.stControlPad.bPrepareSequenceStateInvisible := FALSE;
					iq_stVisControl.stControlPad.bStateSignalPrepareYellow      := TRUE;
		ELSIF iq_XTags.Status = E_XMotion_Status.Prepared THEN
					iq_stVisControl.stControlPad.bStateSignalPrepareGreen := TRUE;
		ELSIF iq_XTags.Status = E_XMotion_Status.Execute THEN
					iq_stVisControl.stControlPad.bStartSequenceStateInvisible := FALSE;
					iq_stVisControl.stControlPad.bStateSignalExecuteGreen     := TRUE;
		ELSIF iq_XTags.Status = E_XMotion_Status.StartUp THEN
					iq_stVisControl.stControlPad.bStateSignalAbortBlue := TRUE;
		END_IF	

	END_IF
END_ACTION

END_FUNCTION_BLOCK

// ---- 1_Industry/FB_VisControl.TcPOU
FUNCTION_BLOCK FB_VisControl

VAR_IN_OUT

	iq_stVisControl  : ST_VisControl;
	iq_XTags		 : ST_XTags;
		
END_VAR


VAR
		
	diStatusOld : DINT := -1;

END_VAR




	// Setting XTag-Commands according to user-commands
	IF    iq_stVisControl.stControlPad.bButtonState_Abort THEN
				iq_XTags.Command  := E_XMotion_Command.Abort;	
	ELSIF iq_stVisControl.stControlPad.bButtonState_Reset THEN
				iq_XTags.Command  := E_XMotion_Command.Reset;	
	ELSIF iq_stVisControl.stControlPad.bButtonState_Prepare THEN
				iq_XTags.Command  := E_XMotion_Command.Prepare;	
	ELSIF iq_stVisControl.stControlPad.bButtonState_Start THEN
				iq_XTags.Command  := E_XMotion_Command.Start;	
	ELSE
				iq_XTags.Command  := E_XMotion_Command.NoCommand;
	END_IF


	
	// Setting Vis display according to current status
	IF iq_XTags.Status <> diStatusOld THEN
		diStatusOld := iq_XTags.Status;	
	
		iq_stVisControl.stControlPad.bStateSignalAbortBlue     := FALSE;
		iq_stVisControl.stControlPad.bStateSignalAbortYellow   := FALSE;
		iq_stVisControl.stControlPad.bStateSignalAbortGreen    := FALSE;
		iq_stVisControl.stControlPad.bStateSignalResetYellow   := FALSE;
		iq_stVisControl.stControlPad.bStateSignalResetGreen    := FALSE;		
		iq_stVisControl.stControlPad.bStateSignalResetYellow   := FALSE;
		iq_stVisControl.stControlPad.bStateSignalResetGreen    := FALSE;		
		iq_stVisControl.stControlPad.bStateSignalPrepareYellow := FALSE;
		iq_stVisControl.stControlPad.bStateSignalPrepareGreen  := FALSE;		
		iq_stVisControl.stControlPad.bStateSignalExecuteYellow := FALSE;
		iq_stVisControl.stControlPad.bStateSignalExecuteGreen  := FALSE;	

		IF 	   iq_XTags.Status = E_XMotion_Status.Aborting THEN
					iq_stVisControl.stControlPad.bStateSignalAbortYellow   := TRUE;		
		ELSIF iq_XTags.Status = E_XMotion_Status.Aborted THEN
					iq_stVisControl.stControlPad.bStateSignalAbortGreen    := TRUE;
		ELSIF iq_XTags.Status = E_XMotion_Status.Resetting THEN
					iq_stVisControl.stControlPad.bStateSignalResetYellow   := TRUE;
		ELSIF iq_XTags.Status = E_XMotion_Status.Stopped THEN
					iq_stVisControl.stControlPad.bStateSignalResetGreen    := TRUE;
		ELSIF iq_XTags.Status = E_XMotion_Status.Preparing THEN
					iq_stVisControl.stControlPad.bStateSignalPrepareYellow := TRUE;
		ELSIF iq_XTags.Status = E_XMotion_Status.Prepared THEN
					iq_stVisControl.stControlPad.bStateSignalPrepareGreen  := TRUE;
		ELSIF iq_XTags.Status = E_XMotion_Status.Execute THEN
					iq_stVisControl.stControlPad.bStateSignalExecuteGreen  := TRUE;
		ELSIF iq_XTags.Status = E_XMotion_Status.StartUp THEN
					iq_stVisControl.stControlPad.bStateSignalAbortBlue     := TRUE;
		END_IF	

	END_IF

END_FUNCTION_BLOCK

// ---- 2_Application/Station/Templates/FB_Station_xx_SW_Separate.TcPOU
FUNCTION_BLOCK FB_Station_xx_SW_Separate EXTENDS FB_StationBase
VAR_INPUT
END_VAR
VAR_OUTPUT
END_VAR

METHOD ClearList : BOOL
VAR_INPUT
END_VAR
SUPER^.ClearList();
// Add aditional Data to Clear in Reset
// List and State will be cleared in master class
ClearList := TRUE;
END_METHOD

METHOD Processing : BOOL
VAR_INPUT
	i_nMachineState 	: INT;		// 1=starting, 2=Running
END_VAR


VAR_INST
	nMoverIndex						: UINT;
	fPositionOnTrack				: LREAL;
	nCurrentTrackIndex				: UDINT;
	fStationPositionOnTrack			: LREAL;
	nStationIndex					: UINT;
	
	nTrackNextStationPositionB		: UINT;
	nTrackNextStationPositionC		: UINT;	
	nNextStationIndexOutputB		: UINT;
	nNextStationIndexOutputC		: UINT;
	nTrackIndexOutputB				: UINT;
	nTrackIndexOutputC				: UINT;
	fSendAwayPositionOutputB		: LREAL;
	fSendAwayPositionOutputC		: LREAL;
	nNextStationIndex				: UINT;
	bSendToOutputB					: BOOL;
	bSendToOutputC					: BOOL;	
	fOutOfRangePosition				: LREAL;
	fMoverSpace						: LREAL;
	
	ClearTrig						: R_TRIG;
		
	nTrackindex						: UINT;
	fMoverPosition					: LREAL;
	fMoverVelocity					: LREAL;
	fMoverAcceleration				: LREAL;
	fMoverJerk						: LREAL;
	strInfo							: STRING;
	
	nErrorId						: UDINT;
	nObjectID						: UDINT;
	nObjectType						: UDINT;	
	
	nDestinationProcess				: UINT;
	nIncommingTrackOID				: UDINT;
			 
END_VAR

// Station - Switch-Seperate


ClearTrig(CLK:=bClearStation);
IF ClearTrig.Q THEN
	nState := 10;	
END_IF

CASE nState OF
	

	0:	// Waiting for initialization
		nState := 10;


	10:	// Init Station Parameters
				   nStationIndex := 0;		// ***HINT*** Station-Paramater to be defined 		
		nNextStationIndexOutputB := 0;		// ***HINT*** Station-Paramater to be defined 
			  nTrackIndexOutputB := 0;		// ***HINT*** Station-Paramater to be defined 
		nNextStationIndexOutputC := 0;		// ***HINT*** Station-Paramater to be defined 
			  nTrackIndexOutputC := 0;		// ***HINT*** Station-Paramater to be defined 
			    	 fMoverSpace := 0;		// ***HINT*** Station-Paramater to be defined 
	    fSendAwayPositionOutputB := 0;		// ***HINT*** Station-Paramater to be defined 
		fSendAwayPositionOutputC := 0;		// ***HINT*** Station-Paramater to be defined 
			
		bClearStation := FALSE;
			   nState := 11;
	
	11: // Fail-safe check, just to make sure all variables have been assigned after doing copy&paste from the template	
		IF             nStationIndex > 0
		AND nNextStationIndexOutputB > 0
		AND       nTrackIndexOutputB > 0
		AND nNextStationIndexOutputC > 0 
		AND       nTrackIndexOutputC > 0 
		AND              fMoverSpace > 0
		AND fSendAwayPositionOutputB > 0
		AND fSendAwayPositionOutputC > 0
		AND              fMoverSpace > 0
		THEN
			nState := 20;
		END_IF

		
	20:	// Calculating station x-y-position 
		PositionOnTrack.fPositionOnTrack := 0.0;
		PositionOnTrack.nTrackId		 := UINT_TO_INT(nTrackIndexOutputB);
		ipTrack[PositionOnTrack.nTrackId].std.GetMoverPositionAt(PositionOnTrack.fPositionOnTrack, StationPosition);
		VisuPosX := StationPosition.x;
		VisuPosY := StationPosition.y;
		nState := 100;

			
	100: // Waiting for Mover
			IF P_List.P_FirstInList <> 0 THEN
				nMoverIndex := P_List.P_FirstInList.P_Id;
				nState := 110;
			END_IF
	
	
	110: // Decide to which Station the mover has to travel to next.	
			nDestinationProcess := ipMoverApplication[nMoverIndex].ProductData.nDestinationProcess;	
			nIncommingTrackOID	:= ipMoverApplication[nMoverIndex].std.P_SetOnTrack.TrackOID;
			nTrackindex := 0;
						
			CASE nDestinationProcess OF
			0: // -> OutputB
				nNextStationIndex  := nNextStationIndexOutputB;
				fMoverPosition     := fSendAwayPositionOutputB;
				nTrackindex        := nTrackIndexOutputB;		
		
			2: // -> OutputC
				nNextStationIndex  := nNextStationIndexOutputC;
				fMoverPosition     := fSendAwayPositionOutputC;
				nTrackindex        := nTrackIndexOutputC;				
	
			3: // -> OutputB
				nNextStationIndex  := nNextStationIndexOutputB;
				fMoverPosition     := fSendAwayPositionOutputB;
				nTrackindex        := nTrackIndexOutputB;		
			END_CASE
			
			IF nTrackindex > 0 THEN
				nState := 200;	
			END_IF


		

	200: 	// Send mover to the next station
			fMoverVelocity     :=    300.0;
			fMoverAcceleration :=  1_000.0;
			fMoverJerk         := 10_000.0;	
	
			stMoveParameters.direction := Tc3_Mc3PlanarMotion.MC_DIRECTION.mcDirectionPositive;
			stMoveParameters.gap       := 240.0;
		
			strInfo := CONCAT('Station: ', UINT_TO_STRING(nStationIndex));
			strInfo := CONCAT(strInfo, ' move to next Station:' );
			strInfo := CONCAT(strInfo, UINT_TO_STRING(nNextStationIndex));
		
	
			IF NOT ipMoverApplication[nMoverIndex].std.P_MoveOnTrack.Error THEN

				FOR idx:=10 TO 1 BY -1 DO 
					strInfoHistory[idx] := strInfoHistory[idx-1];
				END_FOR
				strInfoHistory[0] := strInfo;

		
				ipMoverApplication[nMoverIndex].std.MoveOnTrack( strInfo,
																 ipTrack[nTrackindex].std,
																 fMoverPosition,
																 fMoverVelocity,
																 fMoverAcceleration,
																 fMoverJerk,
																 stMoveParameters.gap,
																 stMoveParameters.direction);
																 																			 
		   		 nState := nState +1;
				 
			ELSIF ipMoverApplication[nMoverIndex].std.P_MoveOnTrack.Error THEN
				   nErrorID := ipMoverApplication[nMoverIndex].std.P_MoveOnTrack.ErrorID;
				  nObjectID := ipMoverApplication[nMoverIndex].std.P_MoveOnTrack.stInfo.nObjectID;
				nObjectType := ipMoverApplication[nMoverIndex].std.P_MoveOnTrack.stInfo.nObjectType;				
			END_IF
		

			
	201: 	IF ipMoverApplication[nMoverIndex].std.P_MoveOnTrack.Active
			OR ipMoverApplication[nMoverIndex].std.P_MoveOnTrack.Done 
			THEN
				nState := 210;
				
			ELSIF ipMoverApplication[nMoverIndex].std.P_MoveOnTrack.Error THEN
				
				   nErrorID := ipMoverApplication[nMoverIndex].std.P_MoveOnTrack.ErrorID;
				  nObjectID := ipMoverApplication[nMoverIndex].std.P_MoveOnTrack.stInfo.nObjectID;
				nObjectType := ipMoverApplication[nMoverIndex].std.P_MoveOnTrack.stInfo.nObjectType;
			END_IF			
	

	210: // Check if Mover passed the junction point		
			IF ipMoverApplication[nMoverIndex].std.P_SetOnTrack.TrackOID <> nIncommingTrackOID THEN 
				nState := 220;
			END_IF

	
	220: // Mover to the list of the next station
		ipStation[nNextStationIndex].P_List.AddMover(P_List.RemoveFirstInList());
		nState := 500;	
	
		
	500: // done for this cycle
		nState := 100;

END_CASE
END_METHOD

END_FUNCTION_BLOCK

// ---- 2_Application/Station/Templates/FB_Station_xx_SW_Merge.TcPOU
FUNCTION_BLOCK FB_Station_xx_SW_Merge EXTENDS FB_StationBase
VAR_INPUT
END_VAR
VAR_OUTPUT
END_VAR

METHOD ClearList : BOOL
VAR_INPUT
END_VAR
SUPER^.ClearList();
// Add aditional Data to Clear in Reset
// List and State will be cleared in master class
ClearList := TRUE;
END_METHOD

METHOD Processing : BOOL
VAR_INPUT
	i_nMachineState 	: INT;		// 1=Starting, 2=Running
END_VAR

VAR_INST
	
	ClearTrig					: R_TRIG;
	
	fStationPositionOnTrack		: LREAL;

	nStationIndex				: UINT;
	nNextStationIndex			: UINT;
	nNextStationTrackIndex		: UINT;
	nMoverIndex					: UINT;
	nNextStationIndexOutputA	: UINT;
	nTrackIndexOutputA			: UINT;	
	fSendAwayPositionOutputA	: LREAL;	

	nMoverIndexInputB			: UINT;
	nMoverIndexInputC			: UINT;
	nTrackIndex					: UINT;
	fMoverPosition				: LREAL;
	fMoverVelocity				: LREAL;
	fMoverAcceleration			: LREAL;
	fMoverJerk					: LREAL;
	nIncommingTrackOID			: UDINT;
	
	nErrorId					: UDINT;
	nObjectID					: UDINT;
	nObjectType					: UDINT;	
	
END_VAR

// Station - Switch-Merge	


ClearTrig(CLK:=bClearStation);
IF ClearTrig.Q THEN
	nState := 10;	
END_IF

CASE nState OF
	
	0:	// Waiting for initialization
		nState := 10;
	

	
	10:	// Init Station-Parameters	
					   nStationIndex := 0;		
			nNextStationIndexOutputA := 0;	
				  nTrackIndexOutputA := 0;		
			fSendAwayPositionOutputA := 0.0;			
				
			bClearStation := FALSE;
			       nState := 11;

	11: // Fail-safe check, just to make sure all variables have been assigned after doing copy&paste from the template
		IF             nStationIndex > 0
		AND nNextStationIndexOutputA > 0
		AND       nTrackIndexOutputA > 0
		AND fSendAwayPositionOutputA > 0 
		THEN
			nState := 20;
		END_IF

		
	20:	// Calculating station x-y-position 
		PositionOnTrack.fPositionOnTrack := 0.0;
		PositionOnTrack.nTrackId		 := UINT_TO_INT(nTrackIndexOutputA);
		ipTrack[PositionOnTrack.nTrackId].std.GetMoverPositionAt(PositionOnTrack.fPositionOnTrack, StationPosition);
		VisuPosX := StationPosition.x;
		VisuPosY := StationPosition.y;
		nState := 100;
			   
		
	100: // Waiting for Mover on Input_B or Input_C
		IF P_List.P_FirstInList = 0 THEN
			nMoverIndexInputB := 0;
			nMoverIndexInputC := 0;
		
			IF P_List_Input_B.P_FirstInList <> 0 THEN
				nMoverIndexInputB := P_List_Input_B.P_FirstInList.P_Id;
			END_IF		
			
			IF P_List_Input_C.P_FirstInList <> 0 THEN
				nMoverIndexInputC := P_List_Input_C.P_FirstInList.P_Id;
			END_IF				
			
			IF nMoverIndexInputB > 0 
			OR nMoverIndexInputC > 0
			THEN
				 nState := 110;
			END_IF
		ELSE
			nState := 120;
		END_IF
		
		
	110: // Priority: B comes first  
		IF nMoverIndexInputB > 0 THEN
			P_List.AddMover(P_List_Input_B.RemoveFirstInList());
		ELSE
			P_List.AddMover(P_List_Input_C.RemoveFirstInList());
		END_IF	
		nState := 120;
		
		
	120: // Processing mover to next Station
		IF P_List.P_FirstInList <> 0 THEN
			       nMoverIndex := P_List.P_FirstInList.P_Id;
			nIncommingTrackOID := ipMoverApplication[nMoverIndex].std.P_SetOnTrack.TrackOID;
			            nState := 200;
		END_IF
		
			 
	200: 	// Send mover to the next station output A
			nNextStationIndex  := nNextStationIndexOutputA;
			nTrackIndex 	   := nTrackIndexOutputA;			
			fMoverPosition     := fSendAwayPositionOutputA;
			fMoverVelocity     :=    300.0;
			fMoverAcceleration :=  1_000.0;
			fMoverJerk         := 10_000.0;	
	
			stMoveParameters.direction := Tc3_Mc3PlanarMotion.MC_DIRECTION.mcDirectionPositive;
			stMoveParameters.gap       := 240.0;
		
			strInfo := CONCAT('Station: ', UINT_TO_STRING(nStationIndex));
			strInfo := CONCAT(strInfo, ' move to next Station:' );
			strInfo := CONCAT(strInfo, UINT_TO_STRING(nNextStationIndex));
			

			
	
			IF NOT ipMoverApplication[nMoverIndex].std.P_MoveOnTrack.Error THEN

				FOR idx:=10 TO 1 BY -1 DO 
					strInfoHistory[idx] := strInfoHistory[idx-1];
				END_FOR
				strInfoHistory[0] := strInfo;				

				ipMoverApplication[nMoverIndex].std.MoveOnTrack( strInfo,
																 ipTrack[nTrackIndex].std,
																 fMoverPosition,
																 fMoverVelocity,
																 fMoverAcceleration,
																 fMoverJerk,
																 stMoveParameters.gap,
																 stMoveParameters.direction);
																 
																 
			ipMoverApplication[nMoverIndex].P_nTrackId := nNextStationTrackIndex;
															 
		    nState := nState +1;
			
			ELSIF ipMoverApplication[nMoverIndex].std.P_MoveOnTrack.Error THEN
				   nErrorID := ipMoverApplication[nMoverIndex].std.P_MoveOnTrack.ErrorID;
				  nObjectID := ipMoverApplication[nMoverIndex].std.P_MoveOnTrack.stInfo.nObjectID;
				nObjectType := ipMoverApplication[nMoverIndex].std.P_MoveOnTrack.stInfo.nObjectType;				
			END_IF			
			

	201: 	IF ipMoverApplication[nMoverIndex].std.P_MoveOnTrack.Error THEN
				   nErrorID := ipMoverApplication[nMoverIndex].std.P_MoveOnTrack.ErrorID;
				  nObjectID := ipMoverApplication[nMoverIndex].std.P_MoveOnTrack.stInfo.nObjectID;
				nObjectType := ipMoverApplication[nMoverIndex].std.P_MoveOnTrack.stInfo.nObjectType;		
			ELSE
				IF ipMoverApplication[nMoverIndex].std.P_MoveOnTrack.Active 
				OR ipMoverApplication[nMoverIndex].std.P_MoveOnTrack.Done
				THEN
					nState := 210;
				END_IF
			END_IF

			
	210: // Check if Mover passed the junction point		
		IF ipMoverApplication[nMoverIndex].std.P_SetOnTrack.TrackOID <> nIncommingTrackOID THEN 
			nState := 220;
		END_IF
	
	
	220: // Check if Mover is out of range
		IF ipMoverApplication[nMoverIndex].std.P_SetOnTrack.SetPos > 120.0 THEN 
			nState := 230;
		END_IF

	
	230: // Mover to the list of the next station
		ipStation[nNextStationIndex].P_List.AddMover(P_List.RemoveFirstInList());
		nState := 500;	
	
		
	500: // done for this cycle
		nState := 100;
		
	
END_CASE
END_METHOD

END_FUNCTION_BLOCK

// ---- 2_Application/Station/Templates/FB_Station_xx_Process.TcPOU
FUNCTION_BLOCK FB_Station_xx_Process EXTENDS FB_StationBase
VAR_INPUT
END_VAR
VAR_OUTPUT
END_VAR
VAR
END_VAR

METHOD ClearList : BOOL
VAR_INPUT
END_VAR
SUPER^.ClearList();
// Add aditional Data to Clear in Reset
// List and State will be cleared in master class
ClearList := TRUE;
END_METHOD

METHOD Processing : BOOL
VAR_INPUT
	i_nMachineState 	: INT;		// 1=starting, 2=Running
END_VAR



VAR_INST

	bToggleSwitch	: BOOL;
	bStationActive				: BOOL;

	nMoverIndex					: UINT;
	fPositionOnTrack			: LREAL;
	nCurrentTrackIndex			: UDINT;
	
	nStationIndex				: UINT;
	nNextStationIndex			: UINT;
	nStationTrackIndex			: UINT;
	fStationPositionOnTrack		: LREAL;
	fSendAwayPosition			: LREAL;
	fInRangePosition			: LREAL;
	fOutOfRangePosition			: LREAL;
	
	fMoverPosition				: LREAL;
	nTrackIndex					: UINT;
	fMoverVelocity				: LREAL;
	fMoverAcceleration			: LREAL;
	fMoverJerk					: LREAL;
	strInfo						: STRING;
	
	nErrorId					: UDINT;
	nObjectID					: UDINT;
	nObjectType					: UDINT;						
	
	Timer01						: TON;
	ClearTrig					: R_TRIG;
	
	TrackInfo					: PlanarObjectInfo;
	nStationTrackID				: UDINT;
	nMoverOnTrackID				: UDINT;
	
END_VAR


// *** Processing Station ***

ClearTrig(CLK:=bClearStation);
IF ClearTrig.Q THEN
	nState := 10;	
END_IF


CASE nState OF

	0:		// Waiting for initialization	
			nState := 10;

	10:		// Init Station-Parameters				
				      nStationIndex := 0;	// ***HINT*** Station-Paramater to be defined 
			     nStationTrackIndex := 0;	// ***HINT*** Station-Paramater to be defined 
			      nNextStationIndex := 0;	// ***HINT*** Station-Paramater to be defined 
			fStationPositionOnTrack := 0;	// ***HINT*** Station-Paramater to be defined 
				  fSendAwayPosition := 0; 	// ***HINT*** Station-Paramater to be defined 
										
			bClearStation := FALSE;
				   nState := 11;

	11: // Fail-safe check, just to make sure all variables have been assigned after doing copy&paste from the template
			IF            nStationIndex > 0
			AND      nStationTrackIndex > 0
			AND       nNextStationIndex > 0
			AND fStationPositionOnTrack > 0
			AND       fSendAwayPosition > 0
			THEN   
				nState := 20;
			END_IF
			
				   
	20:		// Calculating station x-y-position 
			PositionOnTrack.fPositionOnTrack := fStationPositionOnTrack;
 			PositionOnTrack.nTrackId		 := UINT_TO_INT(nStationTrackIndex);
			ipTrack[PositionOnTrack.nTrackId].std.GetMoverPositionAt(PositionOnTrack.fPositionOnTrack, StationPosition);
			VisuPosX := StationPosition.x;
			VisuPosY := StationPosition.y;
			nState := 100;

		
	100: 	// Waiting for Mover
			IF P_List.P_FirstInList <> 0 THEN
					   nMoverIndex := P_List.P_FirstInList.P_Id;
							nState := 110;
			END_IF
	
		
	110: 	// Check if Mover is in range
			TrackInfo := ipTrack[nStationTrackIndex].std.P_Info;
			nStationTrackID := TrackInfo.Id;
			nMoverOnTrackID := ipMoverApplication[nMoverIndex].std.P_SetOnTrack.TrackOID;
			IF nStationTrackID = nMoverOnTrackID  THEN
				nCurrentTrackIndex := nMoverOnTrackID;
							nState := 120;		
			ELSE
				nState := 100;
			END_IF
		
		
	120: 	// Checking product properties
			IF i_nMachineState = 1  THEN    // 1=starting, 2=Running
				IF nStationIndex = 1 THEN
					ipMoverApplication[nMoverIndex].ProductData.bInitRun := FALSE;
				ELSE
					nState := 220;
				END_IF
			ELSIF i_nMachineState = 2 THEN  // 1=starting, 2=Running
				nState := 200;
			ELSE
				nState := 20;	
			END_IF			
		
		
	200: 	// Send mover to Processing-Position
			fMoverPosition     := fStationPositionOnTrack;
			nTrackIndex        := nStationTrackIndex;
			fMoverVelocity     :=    300.0;
			fMoverAcceleration :=  1_000.0;
			fMoverJerk         := 10_000.0;	
	
			stMoveParameters.direction := Tc3_Mc3PlanarMotion.MC_DIRECTION.mcDirectionPositive;
			stMoveParameters.gap       := 240.0;
		
			strInfo := CONCAT('Station: ', UINT_TO_STRING(nStationIndex));
			strInfo := CONCAT(strInfo, ' to processing position');

			
			IF NOT ipMoverApplication[nMoverIndex].std.P_MoveOnTrack.Error THEN
	
				FOR idx:=10 TO 1 BY -1 DO 
					strInfoHistory[idx] := strInfoHistory[idx-1];
				END_FOR
				strInfoHistory[0] := strInfo;		

	
				ipMoverApplication[nMoverIndex].std.MoveOnTrack( strInfo,
																 ipTrack[nTrackIndex].std,
																 fMoverPosition,
																 fMoverVelocity,
																 fMoverAcceleration,
																 fMoverJerk,
																 stMoveParameters.gap,
																 stMoveParameters.direction);
				nState := nState +1;
				
			ELSIF ipMoverApplication[nMoverIndex].std.P_MoveOnTrack.Error THEN
				   nErrorID := ipMoverApplication[nMoverIndex].std.P_MoveOnTrack.ErrorID;
				  nObjectID := ipMoverApplication[nMoverIndex].std.P_MoveOnTrack.stInfo.nObjectID;
				nObjectType := ipMoverApplication[nMoverIndex].std.P_MoveOnTrack.stInfo.nObjectType;				
			END_IF
		
		
	201: 	IF ipMoverApplication[nMoverIndex].std.P_MoveOnTrack.Done THEN
				nState := 210;
			ELSIF ipMoverApplication[nMoverIndex].std.P_MoveOnTrack.Error THEN
				   nErrorID := ipMoverApplication[nMoverIndex].std.P_MoveOnTrack.ErrorID;
				  nObjectID := ipMoverApplication[nMoverIndex].std.P_MoveOnTrack.stInfo.nObjectID;
				nObjectType := ipMoverApplication[nMoverIndex].std.P_MoveOnTrack.stInfo.nObjectType;
			END_IF		
		
		
	210: 	// do process
			Timer01(IN:=TRUE, PT:=T#1S);
			IF Timer01.Q THEN
				Timer01(IN:=FALSE);	
						
				IF nStationIndex = 1 THEN	
					// Station 1 toggeling mover destination to Station2 or Station3
					IF bToggleSwitch THEN
						ipMoverApplication[nMoverIndex].ProductData.nDestinationProcess := 2;
					ELSE
						ipMoverApplication[nMoverIndex].ProductData.nDestinationProcess := 3;		
					END_IF
					bToggleSwitch := NOT bToggleSwitch;					
				ELSE
					ipMoverApplication[nMoverIndex].ProductData.nDestinationProcess := 1;
				END_IF	
				
				nState := 220;
			END_IF

		
	220: 	// Send mover to the next station
			fMoverPosition     := fSendAwayPosition;	
			nTrackIndex        := nStationTrackIndex;		
			fMoverVelocity     :=    300.0;
			fMoverAcceleration :=  1_000.0;
			fMoverJerk         := 10_000.0;	
	
			stMoveParameters.direction := Tc3_Mc3PlanarMotion.MC_DIRECTION.mcDirectionPositive;
			stMoveParameters.gap       := 240.0;
			
			strInfo := CONCAT('Station: ', UINT_TO_STRING(nStationIndex));
			strInfo := CONCAT(strInfo, ' move to next Station:' );
			strInfo := CONCAT(strInfo, UINT_TO_STRING(nNextStationIndex));

			
			IF ipMoverApplication[nMoverIndex].std.P_MoveOnTrack.Done THEN

				FOR idx:=10 TO 1 BY -1 DO 
					strInfoHistory[idx] := strInfoHistory[idx-1];
				END_FOR
				strInfoHistory[0] := strInfo;		
			
				ipMoverApplication[nMoverIndex].std.MoveOnTrack( strInfo,
																 ipTrack[nTrackIndex].std,
																 fMoverPosition,
																 fMoverVelocity,
																 fMoverAcceleration,
																 fMoverJerk,
																 stMoveParameters.gap,
																 stMoveParameters.direction);
				nState := nState +1;
			END_IF		
		
		
	221: 	IF ipMoverApplication[nMoverIndex].std.P_MoveOnTrack.Active
			OR ipMoverApplication[nMoverIndex].std.P_MoveOnTrack.Done 
			THEN
				nState := 230;
			ELSIF ipMoverApplication[nMoverIndex].std.P_MoveOnTrack.Error THEN
				
				   nErrorID := ipMoverApplication[nMoverIndex].std.P_MoveOnTrack.ErrorID;
				  nObjectID := ipMoverApplication[nMoverIndex].std.P_MoveOnTrack.stInfo.nObjectID;
				nObjectType := ipMoverApplication[nMoverIndex].std.P_MoveOnTrack.stInfo.nObjectType;
			END_IF		
		
			
	230: 	// Mover to the list of the next station
			ipStation[nNextStationIndex].P_List.AddMover(P_List.RemoveFirstInList());
			nState := 500;	
	
		
	500: 	// Done for this cycle
			nState := 100;

END_CASE
END_METHOD

END_FUNCTION_BLOCK

// ---- 2_Application/Tracks/Templates/FB_TrackSegment.TcPOU
FUNCTION_BLOCK FB_TrackSegment EXTENDS FB_TrackBase IMPLEMENTS I_TRACK
VAR_INPUT
END_VAR
VAR_OUTPUT
END_VAR


VAR
	



END_VAR

METHOD Initialize : BOOL
VAR_INPUT
	bExecute 			: BOOL;
END_VAR

VAR_INST
	nState			: INT;
	fbR_TrigExecute : R_TRIG;

	TrackTable		: ARRAY[1..maxNumTrackPoints,1..3] OF LREAL;
	nPointIndex		: INT;
	nPointIndexA	: INT;	
	nPointIndexB	: INT;	
	idx1, idx2		: INT;
	nStartFromTrack	: INT;
	nEndAtTrack		: INT;
	bCloseLoop		: BOOL;	
	
